METHOD CREATE_JOB : BOOL
VAR_INPUT
	_byMbFunction	:	BYTE;
	_wMbAdress		:	WORD;
	_pData			:	POINTER TO BYTE;
	_wQuantity		:	WORD;		
END_VAR
VAR	
	pFbMbJob		:	POINTER TO FB_MBJOB;
END_VAR
IF _pData <> 0 THEN
	IF NOT CHECK_IF_JOB_EXIST(_byMbFunction,_wMbAdress,_pData,_wQuantity) THEN
		pFbMbJob := __NEW(FB_MBJOB);
		IF pFbMbJob <> 0 THEN
			_udiDynMemTemp 			:= _udiDynMemTemp + SIZEOF(FB_MBJOB);
			udiDynMem				:= MAX(udiDynMem,_udiDynMemTemp);
			pFbMbJob^.byMbFunction 	:= _byMbFunction;
			pFbMbJob^.wMbAdress	 	:= _wMbAdress;
			pFbMbJob^.pByte		 	:= _pData;
			pFbMbJob^.wQuantity 	:= _wQuantity;
			ADD_MODBUS_JOB(pFbMbJob^);
			xNoChangeHappen			:= FALSE;
			xConfirmAllJobsDone		:= FALSE;
		END_IF;
	END_IF;
END_IF;
END_METHOD

METHOD DESTROY_JOB : BOOL
VAR_INPUT
	_byMbFunction	:	BYTE;
	_wMbAdress		:	WORD;
	_pData			:	POINTER TO BYTE;
	_wQuantity		:	WORD;		
END_VAR
VAR	
	udiSafe			:	UDINT;
	_TEMP_DES_JOB	:	ITF_MBJOB;
END_VAR
IF __QUERYINTERFACE(_BASE_MBU_JOB,_TEMP_DES_JOB) THEN
	REPEAT 
		IF _TEMP_DES_JOB.byMbFunction = _byMbFunction AND
			_TEMP_DES_JOB.wMbAdress	= _wMbAdress AND
			_TEMP_DES_JOB.pByte = _pData AND
			_TEMP_DES_JOB.wQuantity = _wQuantity THEN
			IF _TEMP_DES_JOB = _TEMP_REG_JOB THEN
				_TEMP_REG_JOB := _TEMP_DES_JOB.BIG_SYBIL;
			END_IF;
			IF _TEMP_DES_JOB = _BASE_MBU_JOB THEN
				_BASE_MBU_JOB := _TEMP_DES_JOB.LOW_SYBIL;
				IF NOT __QUERYINTERFACE(_BASE_MBU_JOB,_BASE_MBU_JOB) THEN
					_TEMP_REG_JOB := _BASE_MBU_JOB;
				END_IF;
			END_IF;
			_TEMP_DES_JOB.DESTROY();
			_COUNT 			:= _COUNT -1;
			_udiDynMemTemp 	:= _udiDynMemTemp - SIZEOF(FB_MBJOB);
			DESTROY_JOB 	:= TRUE;
		ELSE
			_TEMP_DES_JOB := _TEMP_DES_JOB.LOW_SYBIL;
		END_IF;
		udiSafe	:= udiSafe + 1;
	UNTIL DESTROY_JOB OR _TEMP_DES_JOB = 0 OR udiSafe >= 16#FFFFFFFE
	END_REPEAT
ELSE
	DESTROY_JOB := FALSE;
END_IF
END_METHOD

PROPERTY ERROR : BOOL
GET
ERROR := xErrorHappen;
END_GET
SET
xErrorHappen := ERROR;
END_SET
END_PROPERTY

{attribute 'estimated-stack-usage' := '104'}
PROPERTY BIG_SYBIL : ITF_CLIENT
GET
BIG_SYBIL := _ITF_BIG_SYBIL;
END_GET
SET
_ITF_BIG_SYBIL := BIG_SYBIL;
IF __QUERYINTERFACE(_ITF_BIG_SYBIL,_ITF_BIG_SYBIL) THEN
	IF _ITF_BIG_SYBIL.LOW_SYBIL <> SELF THEN
		_ITF_BIG_SYBIL.LOW_SYBIL := THIS^;
	END_IF;
END_IF;
END_SET
END_PROPERTY

METHOD CALL_AFTER_LAST_JOB_DONE
VAR_INPUT
END_VAR
xConfirmAllJobsDone := xNoChangeHappen;
xGetReadyCalled := FALSE;
IF xDestroyAllJobs THEN
	DESTROY_ALL_JOBS();
	xDestroyAllJobs := FALSE;
END_IF;
END_METHOD

METHOD CHECK_IF_JOB_EXIST : BOOL
VAR_INPUT
	_byMbFunction	:	BYTE;
	_wMbAdress		:	WORD;
	_pByte			:	POINTER TO BYTE;
	_wQuantity		:	WORD;	
END_VAR
VAR
	_TEMP_CHK_JOB	:	ITF_MBJOB;
	udiSafe			:	UDINT;
END_VAR
IF __QUERYINTERFACE(_BASE_MBU_JOB,_TEMP_CHK_JOB) THEN
	REPEAT 
		IF _TEMP_CHK_JOB.byMbFunction = _byMbFunction AND
			_TEMP_CHK_JOB.wMbAdress	= _wMbAdress AND
			_TEMP_CHK_JOB.pByte = _pByte AND
			_TEMP_CHK_JOB.wQuantity = _wQuantity THEN
			CHECK_IF_JOB_EXIST := TRUE;
		END_IF;
		_TEMP_CHK_JOB := _TEMP_CHK_JOB.LOW_SYBIL;
		udiSafe	:= udiSafe + 1;
	UNTIL CHECK_IF_JOB_EXIST OR _TEMP_CHK_JOB = 0 OR udiSafe >= 16#FFFFFFFE
	END_REPEAT
ELSE
	CHECK_IF_JOB_EXIST := FALSE;
END_IF
END_METHOD

PROPERTY CONFIRM_ALL_JOBS_DONE : BOOL
GET
CONFIRM_ALL_JOBS_DONE := xConfirmAllJobsDone;
END_GET
END_PROPERTY

PROPERTY AllJobsDone : BOOL
GET
AllJobsDone := xAllJobsDone;
END_GET
END_PROPERTY

PROPERTY AY_ITF_MBJOB_VIS : ARRAY[0..9] OF ITF_MBJOB
GET
AY_ITF_MBJOB_VIS := _ayITF_MBJOB_VIS;
END_GET
END_PROPERTY

PROPERTY BASE_MBJOB : ITF_MBJOB
GET
BASE_MBJOB := _BASE_MBU_JOB;
END_GET
END_PROPERTY

PROPERTY ERROR_ID : ModbusFB.Error
GET
ERROR_ID := eErrorID;
END_GET
SET
eErrorID := ERROR_ID;
END_SET
END_PROPERTY

PROPERTY ExecuteTime : LTIME
GET
ExecuteTime := ltTime;
END_GET
END_PROPERTY

PROPERTY EXEPTION_CODE : ModbusFB.ExceptionCodes
GET
EXEPTION_CODE := eExeptionCode;
END_GET
SET
eExeptionCode := EXEPTION_CODE;
END_SET
END_PROPERTY

METHOD GET_NEXT_JOB : BOOL
VAR_OUTPUT
	_byMbFunction	:	BYTE;
	_wMbAdress		:	WORD;
	_pByte			:	POINTER TO BYTE;
	_wQuantity		:	WORD;	
END_VAR
IF xGetReadyCalled THEN 
	IF __QUERYINTERFACE(_TEMP_MBU_JOB,_TEMP_MBU_JOB) THEN
		_byMbFunction		:= _TEMP_MBU_JOB.byMbFunction;
		_wMbAdress			:= _TEMP_MBU_JOB.wMbAdress;
		_pByte				:= _TEMP_MBU_JOB.pByte;
		_wQuantity			:= _TEMP_MBU_JOB.wQuantity;	
		_TEMP_MBU_JOB		:= _TEMP_MBU_JOB.LOW_SYBIL;
		GET_NEXT_JOB		:= TRUE;
		IF NOT __QUERYINTERFACE(_TEMP_MBU_JOB,_TEMP_MBU_JOB) THEN
			xAllJobsDone 	:= TRUE;
			ltTime			:= fbTimeStop.Stop();
		END_IF;
	ELSIF  __QUERYINTERFACE(_BASE_MBU_JOB,_TEMP_MBU_JOB) THEN 	
		_byMbFunction		:= _TEMP_MBU_JOB.byMbFunction;
		_wMbAdress			:= _TEMP_MBU_JOB.wMbAdress;
		_pByte				:= _TEMP_MBU_JOB.pByte;
		_wQuantity			:= _TEMP_MBU_JOB.wQuantity;
		_TEMP_MBU_JOB		:= _TEMP_MBU_JOB.LOW_SYBIL;
		GET_NEXT_JOB    	:= TRUE;
		fbTimeStop.Start();
	END_IF;
END_IF;
END_METHOD

METHOD GET_READY : BOOL
VAR_INPUT
END_VAR
xGetReadyCalled := TRUE;
xNoChangeHappen := TRUE;
xAllJobsDone	:= FALSE;
_TEMP_MBU_JOB   := 0;
END_METHOD

PROPERTY IsCurrentCall : BOOL
GET
IsCurrentCall := xGetReadyCalled;
END_GET
END_PROPERTY

{attribute 'estimated-stack-usage' := '104'}
PROPERTY LOW_SYBIL : ITF_CLIENT
GET
LOW_SYBIL := _ITF_LOW_SYBIL;
END_GET
SET
_ITF_LOW_SYBIL := LOW_SYBIL;
IF __QUERYINTERFACE(_ITF_LOW_SYBIL,_ITF_LOW_SYBIL) THEN
	IF _ITF_LOW_SYBIL.BIG_SYBIL <> SELF THEN
		_ITF_LOW_SYBIL.BIG_SYBIL := THIS^;
	END_IF;
END_IF;
END_SET
END_PROPERTY

METHOD RELOAD_ARRAY
VAR_INPUT
	xInit				:	BOOL;
	xLoadNext10			:	BOOL;
	xLoadLast10			:	BOOL;
END_VAR
VAR
	diFor				:	DINT;
	ITF_TEMP_MBJOB_VIS	:	ITF_MBJOB;
	ITF_TEMP_SAFE		:	ITF_MBJOB;
	ITF_TEMP_LAST_VALID	:	ITF_MBJOB;
END_VAR
(* Init Array *)
IF xInit THEN
	_ayITF_MBJOB_VIS[LOWER_BOUND(_ayITF_MBJOB_VIS,1)] := _BASE_MBU_JOB;
	FOR diFor := LOWER_BOUND(_ayITF_MBJOB_VIS,1) TO UPPER_BOUND(_ayITF_MBJOB_VIS,1) -1 DO
		IF __QUERYINTERFACE(_ayITF_MBJOB_VIS[diFor],ITF_TEMP_MBJOB_VIS) THEN
			_ayITF_MBJOB_VIS[diFor + 1]	:= _ayITF_MBJOB_VIS[diFor].LOW_SYBIL;
		ELSE
			_ayITF_MBJOB_VIS[diFor + 1] := 0;
		END_IF;	
	END_FOR;
(* Load Next 10 *)
ELSIF xLoadNext10 THEN
	IF __QUERYINTERFACE(_ayITF_MBJOB_VIS[UPPER_BOUND(_ayITF_MBJOB_VIS,1)],ITF_TEMP_MBJOB_VIS) THEN
		_ayITF_MBJOB_VIS[LOWER_BOUND(_ayITF_MBJOB_VIS,1)] := ITF_TEMP_MBJOB_VIS.LOW_SYBIL;
		FOR diFor := LOWER_BOUND(_ayITF_MBJOB_VIS,1) TO UPPER_BOUND(_ayITF_MBJOB_VIS,1) -1 DO
			IF __QUERYINTERFACE(_ayITF_MBJOB_VIS[diFor],ITF_TEMP_MBJOB_VIS) THEN
				_ayITF_MBJOB_VIS[diFor + 1]	:= _ayITF_MBJOB_VIS[diFor].LOW_SYBIL;
			ELSE
				_ayITF_MBJOB_VIS[diFor + 1] := 0;
			END_IF;	
		END_FOR;
	END_IF;
(* Load Last 10 *)
ELSIF xLoadLast10 THEN
	IF __QUERYINTERFACE(_ayITF_MBJOB_VIS[LOWER_BOUND(_ayITF_MBJOB_VIS,1)],ITF_TEMP_MBJOB_VIS) THEN
		IF __QUERYINTERFACE(_ayITF_MBJOB_VIS[LOWER_BOUND(_ayITF_MBJOB_VIS,1)].BIG_SYBIL,ITF_TEMP_SAFE) THEN
			_ayITF_MBJOB_VIS[UPPER_BOUND(_ayITF_MBJOB_VIS,1)] := ITF_TEMP_MBJOB_VIS.BIG_SYBIL;
			FOR diFor := UPPER_BOUND(_ayITF_MBJOB_VIS,1) TO LOWER_BOUND(_ayITF_MBJOB_VIS,1) + 1 BY -1 DO 
				IF __QUERYINTERFACE(_ayITF_MBJOB_VIS[diFor],ITF_TEMP_MBJOB_VIS) THEN
					ITF_TEMP_LAST_VALID  		:= _ayITF_MBJOB_VIS[diFor];
					_ayITF_MBJOB_VIS[diFor - 1]	:= _ayITF_MBJOB_VIS[diFor].BIG_SYBIL;
				ELSE
					(* Resort if new ones Inside *)
					_ayITF_MBJOB_VIS[LOWER_BOUND(_ayITF_MBJOB_VIS,1)] := ITF_TEMP_LAST_VALID;
					FOR diFor := LOWER_BOUND(_ayITF_MBJOB_VIS,1) TO UPPER_BOUND(_ayITF_MBJOB_VIS,1) -1 DO
						IF __QUERYINTERFACE(_ayITF_MBJOB_VIS[diFor],ITF_TEMP_MBJOB_VIS) THEN
							_ayITF_MBJOB_VIS[diFor + 1]	:= _ayITF_MBJOB_VIS[diFor].LOW_SYBIL;
						ELSE
							_ayITF_MBJOB_VIS[diFor + 1] := 0;
						END_IF;	
					END_FOR;					
				END_IF;	
			END_FOR;
		END_IF;
	END_IF;	
END_IF;
END_METHOD

PROPERTY SELF : ITF_CLIENT
GET
SELF := THIS^;
END_GET
END_PROPERTY

METHOD DESTROY_ALL_JOBS_REQUEST
VAR_INPUT
END_VAR
xDestroyAllJobs := TRUE;
END_METHOD

PROPERTY DESTROY_ALL_JOBS_ACTIVE : BOOL
GET
DESTROY_ALL_JOBS_ACTIVE := xDestroyAllJobs;
END_GET
END_PROPERTY

METHOD INTERNAL DESTROY_ALL_JOBS
VAR_INPUT
END_VAR
VAR
	_TEMP_DES_JOB	:	ITF_MBJOB;
	_NEXT_DES_JOB	:	ITF_MBJOB;
	udiSafe			:	UDINT;
END_VAR
IF __QUERYINTERFACE(_BASE_MBU_JOB,_NEXT_DES_JOB) THEN
	_BASE_MBU_JOB := 0;
	_TEMP_REG_JOB := 0;
	_TEMP_MBU_JOB := 0;
	REPEAT 
		IF __QUERYINTERFACE(_NEXT_DES_JOB, _TEMP_DES_JOB) THEN
			_NEXT_DES_JOB := _TEMP_DES_JOB.LOW_SYBIL;
			_TEMP_DES_JOB.DESTROY();
			_COUNT 			:= _COUNT -1;
			_udiDynMemTemp 	:= _udiDynMemTemp - SIZEOF(FB_MBJOB);
		END_IF;
		udiSafe	:= udiSafe + 1;
	UNTIL _NEXT_DES_JOB = 0 OR udiSafe >= 16#FFFFFFFE
	END_REPEAT
END_IF;
END_METHOD

END_FUNCTION_BLOCK

// 30 Program Organization Units/MBJOB/FB_MBJOB
{attribute 'enable_dynamic_creation'}
FUNCTION_BLOCK FB_MBJOB IMPLEMENTS ITF_MBJOB
VAR_OUTPUT
END_VAR
VAR
	_xConfirmExecute:	BOOL;
	_byMbFunction	:	BYTE;
	_wMbAdress		:	WORD;
	_pByte			:	POINTER TO BYTE;
	_wQuantity		:	WORD;	
	_ITF_BIG_SYBIL	:	ITF_MBJOB;
	_ITF_LOW_SYBIL	:	ITF_MBJOB;
	_ITF_PARENT		:	ITF_CLIENT;
END_VAR

PROPERTY wMbAdress : WORD
GET
wMbAdress := _wMbAdress;
END_GET
SET
_wMbAdress := wMbAdress;
END_SET
END_PROPERTY

{attribute 'estimated-stack-usage' := '104'}
PROPERTY BIG_SYBIL : ITF_MBJOB
GET
BIG_SYBIL := _ITF_BIG_SYBIL;
END_GET
SET
_ITF_BIG_SYBIL := BIG_SYBIL;
IF __QUERYINTERFACE(_ITF_BIG_SYBIL,_ITF_BIG_SYBIL) THEN
	IF _ITF_BIG_SYBIL.LOW_SYBIL <> SELF THEN
		_ITF_BIG_SYBIL.LOW_SYBIL := THIS^;
	END_IF;
END_IF;
END_SET
END_PROPERTY

PROPERTY wQuantity : WORD
GET
wQuantity := _wQuantity;
END_GET
SET
_wQuantity := wQuantity;
END_SET
END_PROPERTY

PROPERTY SELF : ITF_MBJOB
GET
SELF := THIS^;
END_GET
END_PROPERTY

PROPERTY byMbFunction : BYTE
SET
_byMbFunction := byMbFunction;
END_SET
GET
byMbFunction := _byMbFunction;
END_GET
END_PROPERTY

METHOD DESTROY
VAR
	pSelf	:	POINTER TO FB_MBJOB;
END_VAR
IF __QUERYINTERFACE(_ITF_BIG_SYBIL,_ITF_BIG_SYBIL) THEN
	_ITF_BIG_SYBIL.LOW_SYBIL := _ITF_LOW_SYBIL;
END_IF;

IF __QUERYINTERFACE(_ITF_LOW_SYBIL,_ITF_LOW_SYBIL) THEN
	_ITF_LOW_SYBIL.BIG_SYBIL := _ITF_BIG_SYBIL;
END_IF;

IF __QUERYINTERFACE(_ITF_PARENT,_ITF_PARENT) THEN
	_ITF_PARENT.RELOAD_ARRAY(TRUE,FALSE,FALSE);
END_IF;

pSelf := THIS;

__DELETE(pSelf);
END_METHOD

{attribute 'estimated-stack-usage' := '104'}
PROPERTY LOW_SYBIL : ITF_MBJOB
SET
_ITF_LOW_SYBIL := LOW_SYBIL;
IF __QUERYINTERFACE(_ITF_LOW_SYBIL,_ITF_LOW_SYBIL) THEN
	IF _ITF_LOW_SYBIL.BIG_SYBIL <> SELF THEN
		_ITF_LOW_SYBIL.BIG_SYBIL := THIS^;
	END_IF;
END_IF;
END_SET
GET
LOW_SYBIL := _ITF_LOW_SYBIL;
END_GET
END_PROPERTY

PROPERTY PARENT : ITF_CLIENT
SET
_ITF_PARENT := PARENT;
END_SET
END_PROPERTY

PROPERTY pByte : POINTER TO BYTE
SET
_pByte := pByte;
END_SET
GET
pByte := _pByte;
END_GET
END_PROPERTY

END_FUNCTION_BLOCK

// 30 Program Organization Units/CLIENTMANAGER/RTU/FB_MB_CLIENTMANAGER_RTU
{attribute 'no_assign'}
FUNCTION_BLOCK FB_MB_CLIENTMANAGER_RTU EXTENDS FB_MB_CLIENTMANAGER IMPLEMENTS ITF_MB_CLIENTMANAGER_RTU
VAR_OUTPUT
END_VAR
VAR
	Client								:	ModbusFB.ClientSerial;
	
	_TEMP_MBU_CLIENT_RTU				:	ITF_MB_CLIENT_RTU;
	
	fbReadCoilsFc01						:	ModbusFB.ClientRequestReadCoils;
	fbReadDiscreteInputsFc02			:	ModbusFB.ClientRequestReadDiscreteInputs;
	fbReadHoldingRegistersFc03			:	ModbusFB.ClientRequestReadHoldingRegisters;
	fbReadInputRegistersFc04			:	ModbusFB.ClientRequestReadInputRegisters;
	fbWriteSingleCoilFc05				:	ModbusFB.ClientRequestWriteSingleCoil;
	fbWriteSingleRegisterFc06			:	ModbusFB.ClientRequestWriteSingleRegister;
	fbWriteMultipleCoilsFc15			:	ModbusFB.ClientRequestWriteMultipleCoils;
	fbWriteMultipleRegistersFc16		:	ModbusFB.ClientRequestWriteMultipleRegisters;
	
	(*Config File *)
	fbConfigFile						:	CtaSysConfig.fbConfigFile;
	scParameter                	 		: 	scSerialPortParameter;
END_VAR

SUPER^();
(* Config *)
actConfig();
(* Check if one is allready Working *)
IF NOT xIsWorking THEN
	(* Get Client Ready *)
	IF __QUERYINTERFACE(_TEMP_MBU_CLIENT,_TEMP_MBU_CLIENT) THEN
		xIsWorking 		:= TRUE;	
		xErrorHappen	:= FALSE;
		eErrorID		:= ModbusFB.Error.OK;
		eExeptionCode	:= ModbusFB.ExceptionCodes.RESPONSE_SUCCESS;	
	(* Get Base Client Ready *)
	ELSIF __QUERYINTERFACE(_BASE_MBU_CLIENT,_TEMP_MBU_CLIENT) THEN
		xIsWorking 		:= TRUE;
		xErrorHappen	:= FALSE;
		eErrorID		:= ModbusFB.Error.OK;
		eExeptionCode	:= ModbusFB.ExceptionCodes.RESPONSE_SUCCESS;
		ltTime := fbTimeStop.Stop();
		fbTimeStop.Start();
	END_IF;
END_IF;
(* Check if is running *)
IF xIsWorking THEN
	IF __QUERYINTERFACE(_TEMP_MBU_CLIENT,_TEMP_MBU_CLIENT) THEN	
		(* Wait until no Execute *)		
		IF 	NOT	fbReadCoilsFc01.xExecute				AND
			NOT	fbReadDiscreteInputsFc02.xExecute	    AND
			NOT	fbReadHoldingRegistersFc03.xExecute     AND
			NOT	fbReadInputRegistersFc04.xExecute	    AND
			NOT	fbWriteSingleCoilFc05.xExecute		    AND
			NOT	fbWriteSingleRegisterFc06.xExecute	    AND
			NOT	fbWriteMultipleCoilsFc15.xExecute	    AND
			NOT	fbWriteMultipleRegistersFc16.xExecute	THEN
			(* Get Type of Port *) 
			IF __QUERYINTERFACE(_TEMP_MBU_CLIENT,_TEMP_MBU_CLIENT_RTU) THEN
				(* Check if Enabled *)
				IF _TEMP_MBU_CLIENT_RTU.ENABLE AND _TEMP_MBU_CLIENT_RTU.COUNT > 0 THEN
					IF NOT _TEMP_MBU_CLIENT_RTU.IsCurrentCall THEN
						_TEMP_MBU_CLIENT_RTU.GET_READY();
					END_IF;
					(* Connect *)
					IF NOT Client.xConnected THEN
						Client.xConnect		:= TRUE;
						Client.iPort		:= scParameter.fbenPort.proValue;
						Client.dwBaudrate	:= scParameter.fbdwBaudrate.proValue;
						Client.byDataBits	:= scParameter.fbbyDataBits.proValue;
						Client.eParity		:= scParameter.fbenParity.proValue;
						Client.eStopBits	:= scParameter.fbenStopBits.proValue;
						Client.eDTRcontrol	:= scParameter.fbenDTRControl.proValue;
						Client.eRTScontrol	:= scParameter.fbenRTSControl.proValue;
						IF scParameter.fbxRtuAscii.proValue THEN
							Client.eRtuAscii	:= ModbusFB.RtuAscii.ASCII;
						ELSE
							Client.eRtuAscii	:= ModbusFB.RtuAscii.RTU;
						END_IF
					END_IF;
					usiNodeId 			:= _TEMP_MBU_CLIENT_RTU.NODE_ID;
					tTimeOut			:= _TEMP_MBU_CLIENT_RTU.TIMEOUT;
					tReadDelay			:= _TEMP_MBU_CLIENT_RTU.READ_DELAY;
					tWriteDelay	 		:= _TEMP_MBU_CLIENT_RTU.WRITE_DELAY;
				ELSE
					xAbort		:= TRUE;
				END_IF;
			ELSE
				xAbort		:= TRUE;				
			END_IF;
			(* Check if Connected *)
			IF Client.xConnected AND NOT xAbort THEN
				(* Get Job *)
				IF NOT xTrig THEN
					xTrig := _TEMP_MBU_CLIENT.GET_NEXT_JOB(_byMbFunction => _byMbFunction,_wMbAdress => _wMbAdress,_pByte => _pByte,_wQuantity => _wQuantity);
				END_IF;
				
				(* Delay Function *)
				actDelays();
				
				(* Execute Function *)
				actExecuteFunction();
				
				(* Resett Timer *)
				IF tonDelay.Q THEN
					tonDelay(IN := FALSE);
					xTrig := FALSE;
				END_IF;
			END_IF;
		ELSE
			(* Check Busy *)
			actCheckBusy();					
		END_IF;
		(* Get Errors *)
		actGetError();
		(* Check if All Job as Done *)
		IF _TEMP_MBU_CLIENT.AllJobsDone OR xAbort THEN
			(* Wait until no Execute *)		
			IF 	NOT xTrig									AND
				NOT	fbReadCoilsFc01.xExecute				AND
				NOT	fbReadDiscreteInputsFc02.xExecute	    AND
				NOT	fbReadHoldingRegistersFc03.xExecute     AND
				NOT	fbReadInputRegistersFc04.xExecute	    AND
				NOT	fbWriteSingleCoilFc05.xExecute		    AND
				NOT	fbWriteSingleRegisterFc06.xExecute	    AND
				NOT	fbWriteMultipleCoilsFc15.xExecute	    AND
				NOT	fbWriteMultipleRegistersFc16.xExecute	THEN
				_TEMP_MBU_CLIENT.CALL_AFTER_LAST_JOB_DONE();
				(* Set Error if Job > 0 *)
				IF _TEMP_MBU_CLIENT.COUNT > 0 THEN
					_TEMP_MBU_CLIENT.ERROR			:= xErrorHappen;
					_TEMP_MBU_CLIENT.ERROR_ID		:= eErrorID;
					_TEMP_MBU_CLIENT.EXEPTION_CODE	:= eExeptionCode;
				END_IF;
				_TEMP_MBU_CLIENT 				:= _TEMP_MBU_CLIENT.LOW_SYBIL;
				xIsWorking						:= FALSE;
				xAbort							:= FALSE;
				_byMbFunction 					:= 0;
				_wMbAdress	  					:= 0;
				_pByte		  					:= 0;
				_wQuantity						:= 0;
			END_IF;
		END_IF;
	END_IF;
END_IF;

(* Call Functions *)
actCallFunctions();

(* Resett Client on Error *)
IF Client.xError AND Client._xConnect THEN
	Client.xConnect := FALSE;
END_IF
(* Call Client *)
Client(udiLogOptions := ModbusFB.LoggingOptions.ServerExceptionReason);

ACTION actCallFunctions:
(* Call *)
fbReadCoilsFc01(				rClient := client);		
fbReadDiscreteInputsFc02(		rClient := Client);  
fbReadHoldingRegistersFc03(		rClient := Client);
fbReadInputRegistersFc04(		rClient := Client);	  
fbWriteSingleCoilFc05(			rClient := Client);	  
fbWriteSingleRegisterFc06(		rClient := Client);  
fbWriteMultipleCoilsFc15(		rClient := Client);  
fbWriteMultipleRegistersFc16(	rClient := Client);
END_ACTION

ACTION actDelays:
(* Delay Read *)
IF _byMbFunction <= 04 THEN
	tonDelay(IN := xTrig,PT := tReadDelay);
(* Delay Write Single *)
ELSIF _byMbFunction >= 5 AND _byMbFunction <= 6 THEN
	tonDelay(IN := xTrig,PT := tWriteDelay); 
(* Delay Write Multiple *)
ELSIF _byMbFunction >= 15 AND _byMbFunction <= 16 THEN
	tonDelay(IN := xTrig,PT := tWriteDelay); 
ELSE 
	tonDelay(IN := xTrig,PT := T#0MS);
END_IF;
END_ACTION

ACTION actConfig:
fbConfigFile();		
scParameter.fbenPort			(_usiParaNr := 1,itfConfigFb := fbconfigFile , _MinInit :=    0,_MaxInit :=    10);
scParameter.fbdwBaudrate		(_usiParaNr := 2,itfConfigFb := fbconfigFile , _MinInit := 4800,_MaxInit := 115200);
scParameter.fbbyDataBits		(_usiParaNr := 3,itfConfigFb := fbconfigFile , _MinInit :=    0,_MaxInit :=     8);
scParameter.fbenParity			(_usiParaNr := 4,itfConfigFb := fbconfigFile , _MinInit :=    0,_MaxInit :=     2);
scParameter.fbenStopBits		(_usiParaNr := 5,itfConfigFb := fbconfigFile , _MinInit :=    1,_MaxInit :=     3);
scParameter.fbenDTRControl		(_usiParaNr := 6,itfConfigFb := fbconfigFile , _MinInit :=    0,_MaxInit :=     2);
scParameter.fbenRTSControl		(_usiParaNr := 7,itfConfigFb := fbconfigFile , _MinInit :=    0,_MaxInit :=     2);
scParameter.fbxRtuAscii			(_usiParaNr := 8,itfConfigFb := fbconfigFile 								 	);

(* Handle on Change *)
IF scParameter.fbenPort.proStateChanged			OR
   scParameter.fbdwBaudrate.proStateChanged	    OR
   scParameter.fbbyDataBits.proStateChanged	    OR
   scParameter.fbenParity.proStateChanged		OR
   scParameter.fbenStopBits.proStateChanged	    OR
   scParameter.fbenDTRControl.proStateChanged	OR
   scParameter.fbenRTSControl.proStateChanged	OR
   scParameter.fbxRtuAscii.proStateChanged		THEN
   Client.xConnect := FALSE;
END_IF;
END_ACTION

ACTION actExecuteFunction:
(* Read Coils *)
IF _byMbFunction = 01 THEN
	fbReadCoilsFc01.udiReplyTimeout					:= TO_UDINT(tTimeOut) * 1000; 
	fbReadCoilsFc01.udiTimeOut						:= 15000000;
	fbReadCoilsFc01.uiUnitId						:= usiNodeId;
	fbReadCoilsFc01.uiStartItem 					:= TO_UINT(_wMbAdress);
	fbReadCoilsFc01.pData 							:= _pByte;
	fbReadCoilsFc01.uiQuantity						:= TO_UINT(_wQuantity);
	fbReadCoilsFc01.xExecute						:= tonDelay.Q;
(* Read Discret Inputs *)                       	
ELSIF _byMbFunction = 02 THEN                   	
	fbReadDiscreteInputsFc02.udiReplyTimeout		:= TO_UDINT(tTimeOut) * 1000; 
	fbReadDiscreteInputsFc02.udiTimeOut				:= 15000000;
	fbReadDiscreteInputsFc02.uiUnitId				:= usiNodeId;
	fbReadDiscreteInputsFc02.uiStartItem			:= TO_UINT(_wMbAdress);
	fbReadDiscreteInputsFc02.pData 					:= _pByte;
	fbReadDiscreteInputsFc02.uiQuantity				:= TO_UINT(_wQuantity);
	fbReadDiscreteInputsFc02.xExecute				:= tonDelay.Q;
(* Read Holding Registers *)                		
ELSIF _byMbFunction = 03 THEN                   	
	fbReadHoldingRegistersFc03.udiReplyTimeout		:= TO_UDINT(tTimeOut) * 1000; 
	fbReadHoldingRegistersFc03.udiTimeOut			:= 15000000;
	fbReadHoldingRegistersFc03.uiUnitId				:= usiNodeId;          	
	fbReadHoldingRegistersFc03.uiStartItem			:= TO_UINT(_wMbAdress);
	fbReadHoldingRegistersFc03.pData 				:= _pByte;
	fbReadHoldingRegistersFc03.uiQuantity			:= TO_UINT(_wQuantity);
	fbReadHoldingRegistersFc03.xExecute				:= tonDelay.Q;			
(* Read Input Registers *)	                		
ELSIF _byMbFunction = 04 THEN                   	
	fbReadInputRegistersFc04.udiReplyTimeout		:= TO_UDINT(tTimeOut) * 1000; 
	fbReadInputRegistersFc04.udiTimeOut				:= 15000000;
	fbReadInputRegistersFc04.uiUnitId				:= usiNodeId;               	
	fbReadInputRegistersFc04.uiStartItem 			:= TO_UINT(_wMbAdress);
	fbReadInputRegistersFc04.pData 					:= _pByte;
	fbReadInputRegistersFc04.uiQuantity				:= TO_UINT(_wQuantity);
	fbReadInputRegistersFc04.xExecute				:= tonDelay.Q;			
(* Write Single Coil *)	                    		
ELSIF _byMbFunction = 05 THEN                   	
	fbWriteSingleCoilFc05.udiReplyTimeout			:= TO_UDINT(tTimeOut) * 1000; 
	fbWriteSingleCoilFc05.udiTimeOut				:= 15000000;
	fbWriteSingleCoilFc05.uiUnitId					:= usiNodeId;            	
	fbWriteSingleCoilFc05.uiItem 					:= TO_UINT(_wMbAdress);
	fbWriteSingleCoilFc05.xValue 					:= FcBytePointToBoolValue(_pByte);
	fbWriteSingleCoilFc05.xExecute					:= tonDelay.Q;		
(* Write Single Register *)                 		
ELSIF _byMbFunction = 06 THEN                   	
	fbWriteSingleRegisterFc06.udiReplyTimeout		:= TO_UDINT(tTimeOut) * 1000;    
	fbWriteSingleRegisterFc06.udiTimeOut			:= 15000000; 
	fbWriteSingleRegisterFc06.uiUnitId				:= usiNodeId;           	
	fbWriteSingleRegisterFc06.uiItem	  			:= TO_UINT(_wMbAdress);
	fbWriteSingleRegisterFc06.uiValue 				:= FcBytePointToWordValue(_pByte);
	fbWriteSingleRegisterFc06.xExecute				:= tonDelay.Q;		
(* Write Multiple Coils *)		            		
ELSIF _byMbFunction = 15 THEN                   	
	fbWriteMultipleCoilsFc15.udiReplyTimeout		:= TO_UDINT(tTimeOut) * 1000;
	fbWriteMultipleCoilsFc15.udiTimeOut				:= 15000000;
	fbWriteMultipleCoilsFc15.uiUnitId				:= usiNodeId;              	
	fbWriteMultipleCoilsFc15.uiStartItem 			:= TO_UINT(_wMbAdress);
	fbWriteMultipleCoilsFc15.pData 					:= _pByte;
	fbWriteMultipleCoilsFc15.uiQuantity				:= TO_UINT(_wQuantity);
	fbWriteMultipleCoilsFc15.xExecute				:= tonDelay.Q;
(* Write Multiple Registers *)                  	
ELSIF _byMbFunction = 16 THEN                   	
	fbWriteMultipleRegistersFc16.udiReplyTimeout	:= TO_UDINT(tTimeOut) * 1000; 
	fbWriteMultipleRegistersFc16.udiTimeOut			:= 15000000;
	fbWriteMultipleRegistersFc16.uiUnitId			:= usiNodeId;    
	fbWriteMultipleRegistersFc16.uiStartItem 		:= TO_UINT(_wMbAdress);
	fbWriteMultipleRegistersFc16.pData 				:= _pByte;
	fbWriteMultipleRegistersFc16.uiQuantity			:= TO_UINT(_wQuantity);
	fbWriteMultipleRegistersFc16.xExecute			:= tonDelay.Q;	
END_IF;
END_ACTION

ACTION actGetError:
(* Client Error *)
IF Client.xError THEN
	xErrorHappen 	:= Client.xError;
	eErrorID		:= Client.eErrorID;
	eExeptionCode	:= ModbusFB.ExceptionCodes.ACKNOWLEDGE;
	xAbort			:= TRUE;
END_IF;
(* Read Coils Fc01 Error *)
IF fbReadCoilsFc01.xError AND NOT xErrorHappen THEN
	xErrorHappen 	:= fbReadCoilsFc01.xError;
	eErrorID		:= fbReadCoilsFc01.eErrorID;
	eExeptionCode	:= fbReadCoilsFc01.eException;
END_IF;
(* Read Discrete Inputs Fc02 Error *)
IF fbReadDiscreteInputsFc02.xError AND NOT xErrorHappen THEN
	xErrorHappen 	:= fbReadDiscreteInputsFc02.xError;
	eErrorID		:= fbReadDiscreteInputsFc02.eErrorID;
	eExeptionCode	:= fbReadDiscreteInputsFc02.eException;
END_IF;
(* Read Holding Registers Fc03 Error *)
IF fbReadHoldingRegistersFc03.xError AND NOT xErrorHappen THEN
	xErrorHappen 	:= fbReadHoldingRegistersFc03.xError;
	eErrorID		:= fbReadHoldingRegistersFc03.eErrorID;
	eExeptionCode	:= fbReadHoldingRegistersFc03.eException;
END_IF;
(* Read Input Registers Fc04 Error *)
IF fbReadInputRegistersFc04.xError AND NOT xErrorHappen THEN
	xErrorHappen 	:= fbReadInputRegistersFc04.xError;
	eErrorID		:= fbReadInputRegistersFc04.eErrorID;
	eExeptionCode	:= fbReadInputRegistersFc04.eException;
END_IF;
(* Write Single Coil Fc05 Error *)
IF fbWriteSingleCoilFc05.xError AND NOT xErrorHappen THEN
	xErrorHappen 	:= fbWriteSingleCoilFc05.xError;
	eErrorID		:= fbWriteSingleCoilFc05.eErrorID;
	eExeptionCode	:= fbWriteSingleCoilFc05.eException;
END_IF;
(* Write Single Register Fc06 Error *)
IF fbWriteSingleRegisterFc06.xError AND NOT xErrorHappen THEN
	xErrorHappen 	:= fbWriteSingleRegisterFc06.xError;
	eErrorID		:= fbWriteSingleRegisterFc06.eErrorID;
	eExeptionCode	:= fbWriteSingleRegisterFc06.eException;
END_IF;		
(* Write Multiple Coils Fc15 Error *)
IF fbWriteMultipleCoilsFc15.xError AND NOT xErrorHappen THEN
	xErrorHappen 	:= fbWriteMultipleCoilsFc15.xError;
	eErrorID		:= fbWriteMultipleCoilsFc15.eErrorID;
	eExeptionCode	:= fbWriteMultipleCoilsFc15.eException;
END_IF;
(* Write Multiple Registers Fc16 Error *)
IF fbWriteMultipleRegistersFc16.xError AND NOT xErrorHappen THEN
	xErrorHappen 	:= fbWriteMultipleRegistersFc16.xError;
	eErrorID		:= fbWriteMultipleRegistersFc16.eErrorID;
	eExeptionCode	:= fbWriteMultipleRegistersFc16.eException;
END_IF;
END_ACTION

PROPERTY P_fbbyDataBits : CtaSysConfig.ITF_DATATYPE
GET
P_fbbyDataBits := scParameter.fbbyDataBits;
END_GET
END_PROPERTY

PROPERTY P_fbdwBaudrate : CtaSysConfig.ITF_DATATYPE
GET
P_fbdwBaudrate := scParameter.fbdwBaudrate;
END_GET
END_PROPERTY

PROPERTY P_fbenDTRControl : CtaSysConfig.ITF_BYTE
GET
P_fbenDTRControl := scParameter.fbenDTRControl;
END_GET
END_PROPERTY

PROPERTY P_fbenParity : CtaSysConfig.ITF_BYTE
GET
P_fbenParity := scParameter.fbenParity;
END_GET
END_PROPERTY

PROPERTY P_fbenRTSControl : CtaSysConfig.ITF_BYTE
GET
P_fbenRTSControl := scParameter.fbenRTSControl;
END_GET
END_PROPERTY

PROPERTY P_fbenStopBits : CtaSysConfig.ITF_BYTE
GET
P_fbenStopBits := scParameter.fbenStopBits;
END_GET
END_PROPERTY

PROPERTY P_fbxRtuAscii : CtaSysConfig.ITF_DATATYPE
GET
P_fbxRtuAscii := scParameter.fbxRtuAscii;
END_GET
END_PROPERTY

PROPERTY P_fbenPort : CtaSysConfig.ITF_INT
GET
P_fbenPort := scParameter.fbenPort;
END_GET
END_PROPERTY

ACTION actCheckBusy:
(* Reset after Busy *)
fbReadCoilsFc01.xExecute				:= fbReadCoilsFc01.xBusy				;
fbReadDiscreteInputsFc02.xExecute	    := fbReadDiscreteInputsFc02.xBusy		;
fbReadHoldingRegistersFc03.xExecute     := fbReadHoldingRegistersFc03.xBusy		;
fbReadInputRegistersFc04.xExecute	    := fbReadInputRegistersFc04.xBusy		;
fbWriteSingleCoilFc05.xExecute		    := fbWriteSingleCoilFc05.xBusy			;
fbWriteSingleRegisterFc06.xExecute	    := fbWriteSingleRegisterFc06.xBusy		;
fbWriteMultipleCoilsFc15.xExecute	    := fbWriteMultipleCoilsFc15.xBusy		;
fbWriteMultipleRegistersFc16.xExecute   := fbWriteMultipleRegistersFc16.xBusy	;
END_ACTION

END_FUNCTION_BLOCK

// 30 Program Organization Units/CLIENT/RTU/FB_MB_CLIENT_RTU
FUNCTION_BLOCK FB_MB_CLIENT_RTU EXTENDS FB_MB_CLIENT IMPLEMENTS ITF_MB_CLIENT_RTU
VAR_OUTPUT
END_VAR
VAR
	(* Config *)
	fbConfigFile				:	CtaSysConfig.fbConfigFile;
	scParameter					:	scSerialClientParameter;
END_VAR

(* Config File *)
actConfig();

ACTION actConfig:
(* Config File *)
fbConfigFile();

scParameter.fbxEnable		(_usiParaNr := 1,itfConfigFb := fbConfigFile										);		
scParameter.fbusiNodeId		(_usiParaNr := 2,itfConfigFb := fbConfigFile,_MinInit := 0	 , _MaxInit := 247		);		
scParameter.fbtTimeOut		(_usiParaNr := 3,itfConfigFb := fbConfigFile,_MinInit := T#0MS, _MaxInit := T#5M 	);		
scParameter.fbtReadDelay	(_usiParaNr := 4,itfConfigFb := fbConfigFile,_MinInit := T#0MS, _MaxInit := T#5M 	);		
scParameter.fbtWriteDelay	(_usiParaNr := 5,itfConfigFb := fbConfigFile,_MinInit := T#0MS, _MaxInit := T#5M 	);
END_ACTION

PROPERTY ENABLE : BOOL
GET
ENABLE := scParameter.fbxEnable.proValue;
END_GET
END_PROPERTY

PROPERTY NODE_ID : USINT
GET
NODE_ID := scParameter.fbusiNodeId.proValue;
END_GET
END_PROPERTY

PROPERTY P_fbtReadDelay : CtaSysConfig.ITF_DATATYPE
GET
P_fbtReadDelay := scParameter.fbtReadDelay;
END_GET
END_PROPERTY

PROPERTY P_fbtTimeOut : CtaSysConfig.ITF_DATATYPE
GET
P_fbtTimeOut := scParameter.fbtTimeOut;
END_GET
END_PROPERTY

PROPERTY P_fbtWriteDelay : CtaSysConfig.ITF_DATATYPE
GET
P_fbtWriteDelay := scParameter.fbtWriteDelay;
END_GET
END_PROPERTY

PROPERTY P_fbusiNodeId : CtaSysConfig.ITF_DATATYPE
GET
P_fbusiNodeId := scParameter.fbusiNodeId;
END_GET
END_PROPERTY

PROPERTY P_fbxEnable : CtaSysConfig.ITF_DATATYPE
GET
P_fbxEnable := scParameter.fbxEnable;
END_GET
END_PROPERTY

PROPERTY READ_DELAY : TIME
GET
READ_DELAY := scParameter.fbtReadDelay.proValue;
END_GET
END_PROPERTY

PROPERTY TIMEOUT : TIME
GET
TIMEOUT := scParameter.fbtTimeOut.proValue;
END_GET
END_PROPERTY

PROPERTY WRITE_DELAY : TIME
GET
WRITE_DELAY := scParameter.fbtWriteDelay.proValue;
END_GET
END_PROPERTY

END_FUNCTION_BLOCK

// 30 Program Organization Units/CLIENT/TCP/FB_MB_CLIENT_TCP
{attribute 'no_assign'}
FUNCTION_BLOCK FB_MB_CLIENT_TCP EXTENDS FB_MB_CLIENT IMPLEMENTS ITF_MB_CLIENT_TCP
VAR_OUTPUT
END_VAR
VAR
	Client						:	ModbusFB.ClientTCP;
	(* Config *)
	fbConfigFile				:	CtaSysConfig.fbConfigFile;
	scParameter                	: 	scTcpClientParameter;
END_VAR

(* Config File *)
actConfig();

(* Resett Client on Error *)
IF (Client.xError AND Client._xConnect) 
	OR NOT ENABLE
	OR scParameter.fbxEnable.proStateChanged		
	OR scParameter.fbuiPort.proStateChanged		
	OR scParameter.fbstIpAdress.proStateChanged	THEN
	Client.xConnect := FALSE;
END_IF

(* Call Client *)
Client(tConnnectTimeOut := T#5S,udiLogOptions := ModbusFB.LoggingOptions.ServerExceptionReason);

ACTION actConfig:
(* Config File *)
fbConfigFile();

scParameter.fbxEnable		(_usiParaNr := 1,itfConfigFb := fbConfigFile										);		
scParameter.fbusiNodeId		(_usiParaNr := 2,itfConfigFb := fbConfigFile,_MinInit := 0	  , _MaxInit := 255		);		
scParameter.fbtTimeOut		(_usiParaNr := 3,itfConfigFb := fbConfigFile,_MinInit := T#0MS, _MaxInit := T#5M 	);		
scParameter.fbtReadDelay	(_usiParaNr := 4,itfConfigFb := fbConfigFile,_MinInit := T#0MS, _MaxInit := T#5M 	);		
scParameter.fbtWriteDelay	(_usiParaNr := 5,itfConfigFb := fbConfigFile,_MinInit := T#0MS, _MaxInit := T#5M 	);	
scParameter.fbuiPort		(_usiParaNr := 6,itfConfigFb := fbConfigFile										);
scParameter.fbstIpAdress	(_usiParaNr := 7,itfConfigFb := fbConfigFile										);

(* Check Ip *)
IF scParameter.fbstIpAdress.proStateChanged THEN
	IF NOT fcCheckIp(scParameter.fbstIPAdress.proValue) THEN
		fcSetInitialIPString(scParameter.fbstIpAdress);
	END_IF;
END_IF;
END_ACTION

PROPERTY ENABLE : BOOL
GET
ENABLE := scParameter.fbxEnable.proValue;
END_GET
END_PROPERTY

PROPERTY IP_ADRESS : STRING(15)
GET
IP_ADRESS := scParameter.fbstIpAdress.proValue;
END_GET
END_PROPERTY

PROPERTY P_fbtTimeOut : CtaSysConfig.ITF_DATATYPE
GET
P_fbtTimeOut := scParameter.fbtTimeOut;
END_GET
END_PROPERTY

PROPERTY P_fbtWriteDelay : CtaSysConfig.ITF_DATATYPE
GET
P_fbtWriteDelay := scParameter.fbtWriteDelay;
END_GET
END_PROPERTY

PROPERTY P_fbuiPort : CtaSysConfig.ITF_DATATYPE
GET
P_fbuiPort := scParameter.fbuiPort;
END_GET
END_PROPERTY

PROPERTY P_fbusiNodeId : CtaSysConfig.ITF_DATATYPE
GET
P_fbusiNodeId := scParameter.fbusiNodeId;
END_GET
END_PROPERTY

PROPERTY P_fbxEnable : CtaSysConfig.ITF_DATATYPE
GET
P_fbxEnable := scParameter.fbxEnable;
END_GET
END_PROPERTY

PROPERTY WRITE_DELAY : TIME
GET
WRITE_DELAY := scParameter.fbtWriteDelay.proValue;
END_GET
END_PROPERTY

PROPERTY PORT : UINT
GET
PORT := scParameter.fbuiPort.proValue;
END_GET
END_PROPERTY

PROPERTY NODE_ID : USINT
GET
NODE_ID := scParameter.fbusiNodeId.proValue;
END_GET
END_PROPERTY

PROPERTY P_fbstIpAdress : CtaSysConfig.ITF_DATATYPE
GET
P_fbstIpAdress := scParameter.fbstIpAdress;
END_GET
END_PROPERTY

PROPERTY READ_DELAY : TIME
GET
READ_DELAY := scParameter.fbtReadDelay.proValue;
END_GET
END_PROPERTY

PROPERTY P_fbtReadDelay : CtaSysConfig.ITF_DATATYPE
GET
P_fbtReadDelay := scParameter.fbtReadDelay;
END_GET
END_PROPERTY

PROPERTY TIMEOUT : TIME
GET
TIMEOUT := scParameter.fbtTimeOut.proValue;
END_GET
END_PROPERTY

METHOD ConnectTcp : BOOL
VAR_INPUT
END_VAR
IF fcCheckIp(IP_ADRESS) THEN
	Client.uiPort 	:= PORT;
	Client.aIPaddr 	:= fcStringIPtoByteArray(IP_ADRESS);
	Client.xConnect	:= TRUE;
	ConnectTcp 		:= TRUE;
ELSE
	ConnectTcp			:= FALSE;
END_IF;
END_METHOD

PROPERTY Connected : BOOL
GET
Connected := Client.xConnected;
END_GET
END_PROPERTY

PROPERTY ClientTcp : REFERENCE TO ModbusFB.Client
GET
ClientTcp REF= Client;
END_GET
END_PROPERTY

END_FUNCTION_BLOCK

// 30 Program Organization Units/CLIENTMANAGER/TCP/FB_MB_CLIENTMANAGER_TCP_1
{attribute 'no_assign'}
FUNCTION_BLOCK FB_MB_CLIENTMANAGER_TCP_1 EXTENDS FB_MB_CLIENTMANAGER IMPLEMENTS ITF_MB_CLIENTMANAGER_TCP
VAR_OUTPUT
END_VAR
VAR
	Client								:	ModbusFB.ClientTCP;

	_TEMP_MBU_CLIENT_TCP				:	ITF_MB_CLIENT_TCP;
	
	fbReadCoilsFc01						:	ModbusFB.ClientRequestReadCoils;
	fbReadDiscreteInputsFc02			:	ModbusFB.ClientRequestReadDiscreteInputs;
	fbReadHoldingRegistersFc03			:	ModbusFB.ClientRequestReadHoldingRegisters;
	fbReadInputRegistersFc04			:	ModbusFB.ClientRequestReadInputRegisters;
	fbWriteSingleCoilFc05				:	ModbusFB.ClientRequestWriteSingleCoil;
	fbWriteSingleRegisterFc06			:	ModbusFB.ClientRequestWriteSingleRegister;
	fbWriteMultipleCoilsFc15			:	ModbusFB.ClientRequestWriteMultipleCoils;
	fbWriteMultipleRegistersFc16		:	ModbusFB.ClientRequestWriteMultipleRegisters;
	
END_VAR

SUPER^();
(* Check if one is allready Working *)
IF NOT xIsWorking THEN
	(* Get Client Ready *)
	IF __QUERYINTERFACE(_TEMP_MBU_CLIENT,_TEMP_MBU_CLIENT) THEN
		xIsWorking 		:= TRUE;	
		xErrorHappen	:= FALSE;
		eErrorID		:= ModbusFB.Error.OK;
		eExeptionCode	:= ModbusFB.ExceptionCodes.RESPONSE_SUCCESS;		
	(* Get Base Client Ready *)
	ELSIF __QUERYINTERFACE(_BASE_MBU_CLIENT,_TEMP_MBU_CLIENT) THEN
		xIsWorking 		:= TRUE;
		xErrorHappen	:= FALSE;
		eErrorID		:= ModbusFB.Error.OK;
		eExeptionCode	:= ModbusFB.ExceptionCodes.RESPONSE_SUCCESS;
		ltTime 			:= fbTimeStop.Stop();
		fbTimeStop.Start();
	END_IF;
END_IF;
(* Check if is running *)
IF xIsWorking THEN
	IF __QUERYINTERFACE(_TEMP_MBU_CLIENT,_TEMP_MBU_CLIENT) THEN	
		(* Wait until no Execute *)		
		IF 	NOT	fbReadCoilsFc01.xExecute				AND
			NOT	fbReadDiscreteInputsFc02.xExecute	    AND
			NOT	fbReadHoldingRegistersFc03.xExecute     AND
			NOT	fbReadInputRegistersFc04.xExecute	    AND
			NOT	fbWriteSingleCoilFc05.xExecute		    AND
			NOT	fbWriteSingleRegisterFc06.xExecute	    AND
			NOT	fbWriteMultipleCoilsFc15.xExecute	    AND
			NOT	fbWriteMultipleRegistersFc16.xExecute	THEN
			(* Get Type of Port *) 
			IF __QUERYINTERFACE(_TEMP_MBU_CLIENT,_TEMP_MBU_CLIENT_TCP) THEN
				(* Check if Enabled *)
				IF _TEMP_MBU_CLIENT_TCP.ENABLE AND _TEMP_MBU_CLIENT_TCP.COUNT > 0 THEN
					IF NOT _TEMP_MBU_CLIENT_TCP.IsCurrentCall THEN
						_TEMP_MBU_CLIENT_TCP.GET_READY();
						tTimeOut		:= _TEMP_MBU_CLIENT_TCP.TIMEOUT;
						tReadDelay		:= _TEMP_MBU_CLIENT_TCP.READ_DELAY;
						tWriteDelay	 	:= _TEMP_MBU_CLIENT_TCP.WRITE_DELAY;
					END_IF;
					(* Connect *)
					IF NOT Client.xConnected THEN
						IF fcCheckIp(_TEMP_MBU_CLIENT_TCP.IP_ADRESS) THEN
							Client.uiPort 	:= _TEMP_MBU_CLIENT_TCP.PORT;
							Client.aIPaddr 	:= fcStringIPtoByteArray(_TEMP_MBU_CLIENT_TCP.IP_ADRESS);
							Client.xConnect	:= TRUE;
							usiNodeId 		:= _TEMP_MBU_CLIENT_TCP.NODE_ID;
						ELSE
							xAbort := TRUE;
						END_IF;
					END_IF;
				ELSE
					xAbort		:= TRUE;
				END_IF;
			ELSE
				xAbort := TRUE;
			END_IF;
			(* Check if Connected *)
			IF Client.xConnected AND NOT xAbort THEN
				(* Get Job *)
				IF NOT xTrig THEN
					xTrig := _TEMP_MBU_CLIENT.GET_NEXT_JOB(_byMbFunction => _byMbFunction,_wMbAdress => _wMbAdress,_pByte => _pByte,_wQuantity => _wQuantity);
				END_IF;
				
				(* Delay Function *)
				actDelays();
				
				(* Execute Function *)
				actExecuteFunction();
				
				(* Resett Timer *)
				IF tonDelay.Q THEN
					tonDelay(IN := FALSE);
					xTrig := FALSE;
				END_IF;
			END_IF;
		ELSE
			(* Check Busy *)
			actCheckBusy();					
		END_IF;
		(* Get Errors *)
		actGetError();
		(* Check if All Job as Done *)
		IF _TEMP_MBU_CLIENT.AllJobsDone OR xAbort THEN
			(* Wait until no Execute *)		
			IF 	NOT	fbReadCoilsFc01.xExecute				AND
				NOT	fbReadDiscreteInputsFc02.xExecute	    AND
				NOT	fbReadHoldingRegistersFc03.xExecute     AND
				NOT	fbReadInputRegistersFc04.xExecute	    AND
				NOT	fbWriteSingleCoilFc05.xExecute		    AND
				NOT	fbWriteSingleRegisterFc06.xExecute	    AND
				NOT	fbWriteMultipleCoilsFc15.xExecute	    AND
				NOT	fbWriteMultipleRegistersFc16.xExecute	THEN
				_TEMP_MBU_CLIENT.CALL_AFTER_LAST_JOB_DONE();
				(* Set Error if Job > 0 *)
				IF _TEMP_MBU_CLIENT.COUNT > 0 THEN
					_TEMP_MBU_CLIENT.ERROR			:= xErrorHappen;
					_TEMP_MBU_CLIENT.ERROR_ID		:= eErrorID;
					_TEMP_MBU_CLIENT.EXEPTION_CODE	:= eExeptionCode;
				END_IF;
				_TEMP_MBU_CLIENT 					:= _TEMP_MBU_CLIENT.LOW_SYBIL;
				
				IF SUPER^.COUNT_ENABLED() = 1 AND NOT xAbort THEN	
					Client.xConnect := Client.xConnect;
				ELSE
					Client.xConnect				:= FALSE;
				END_IF;
				_byMbFunction 					:= 0;
				_wMbAdress	  					:= 0;
				_pByte		  					:= 0;
				_wQuantity						:= 0;
				xIsWorking						:= FALSE;
				xAbort							:= FALSE;
			END_IF;
		END_IF;
	END_IF;
END_IF;

(* Call Functions *)
actCallFunctions();

(* Resett Client on Error *)
IF Client.xError AND Client._xConnect THEN
	Client.xConnect := FALSE;
END_IF
(* Call Client *)
Client(tConnnectTimeOut := T#5S,udiLogOptions := ModbusFB.LoggingOptions.ServerExceptionReason);

ACTION actCallFunctions:
(* Call *)
fbReadCoilsFc01(				rClient := client);		
fbReadDiscreteInputsFc02(		rClient := Client);  
fbReadHoldingRegistersFc03(		rClient := Client);
fbReadInputRegistersFc04(		rClient := Client);	  
fbWriteSingleCoilFc05(			rClient := Client);	  
fbWriteSingleRegisterFc06(		rClient := Client);  
fbWriteMultipleCoilsFc15(		rClient := Client);  
fbWriteMultipleRegistersFc16(	rClient := Client);
END_ACTION

ACTION actCheckBusy:
(* Reset after Busy *)
fbReadCoilsFc01.xExecute				:= fbReadCoilsFc01.xBusy				;
fbReadDiscreteInputsFc02.xExecute	    := fbReadDiscreteInputsFc02.xBusy		;
fbReadHoldingRegistersFc03.xExecute     := fbReadHoldingRegistersFc03.xBusy		;
fbReadInputRegistersFc04.xExecute	    := fbReadInputRegistersFc04.xBusy		;
fbWriteSingleCoilFc05.xExecute		    := fbWriteSingleCoilFc05.xBusy			;
fbWriteSingleRegisterFc06.xExecute	    := fbWriteSingleRegisterFc06.xBusy		;
fbWriteMultipleCoilsFc15.xExecute	    := fbWriteMultipleCoilsFc15.xBusy		;
fbWriteMultipleRegistersFc16.xExecute   := fbWriteMultipleRegistersFc16.xBusy	;
END_ACTION

ACTION actDelays:
(* Delay Read *)
IF _byMbFunction <= 04 THEN
	tonDelay(IN := xTrig,PT := tReadDelay);
(* Delay Write Single *)
ELSIF _byMbFunction >= 5 AND _byMbFunction <= 6 THEN
	tonDelay(IN := xTrig,PT := tWriteDelay); 
(* Delay Write Multiple *)
ELSIF _byMbFunction >= 15 AND _byMbFunction <= 16 THEN
	tonDelay(IN := xTrig,PT := tWriteDelay); 
ELSE 
	tonDelay(IN := xTrig,PT := T#0MS);
END_IF;
END_ACTION

ACTION actExecuteFunction:
(* Read Coils *)
IF _byMbFunction = 01 THEN
	fbReadCoilsFc01.udiReplyTimeout					:= TO_UDINT(tTimeOut) * 1000; 
	fbReadCoilsFc01.udiTimeOut						:= TO_UDINT(tTimeOut) * 1000 * 2;
	fbReadCoilsFc01.uiUnitId						:= usiNodeId;
	fbReadCoilsFc01.uiStartItem 					:= TO_UINT(_wMbAdress);
	fbReadCoilsFc01.pData 							:= _pByte;
	fbReadCoilsFc01.uiQuantity						:= TO_UINT(_wQuantity);
	fbReadCoilsFc01.xExecute						:= tonDelay.Q;
(* Read Discret Inputs *)                       	
ELSIF _byMbFunction = 02 THEN                   	
	fbReadDiscreteInputsFc02.udiReplyTimeout		:= TO_UDINT(tTimeOut) * 1000; 
	fbReadDiscreteInputsFc02.udiTimeOut				:= TO_UDINT(tTimeOut) * 1000 * 2;
	fbReadDiscreteInputsFc02.uiUnitId				:= usiNodeId;
	fbReadDiscreteInputsFc02.uiStartItem			:= TO_UINT(_wMbAdress);
	fbReadDiscreteInputsFc02.pData 					:= _pByte;
	fbReadDiscreteInputsFc02.uiQuantity				:= TO_UINT(_wQuantity);
	fbReadDiscreteInputsFc02.xExecute				:= tonDelay.Q;
(* Read Holding Registers *)                		
ELSIF _byMbFunction = 03 THEN                   	
	fbReadHoldingRegistersFc03.udiReplyTimeout		:= TO_UDINT(tTimeOut) * 1000; 
	fbReadHoldingRegistersFc03.udiTimeOut			:= TO_UDINT(tTimeOut) * 1000 * 2;
	fbReadHoldingRegistersFc03.uiUnitId				:= usiNodeId;          	
	fbReadHoldingRegistersFc03.uiStartItem			:= TO_UINT(_wMbAdress);
	fbReadHoldingRegistersFc03.pData 				:= _pByte;
	fbReadHoldingRegistersFc03.uiQuantity			:= TO_UINT(_wQuantity);
	fbReadHoldingRegistersFc03.xExecute				:= tonDelay.Q;			
(* Read Input Registers *)	                		
ELSIF _byMbFunction = 04 THEN                   	
	fbReadInputRegistersFc04.udiReplyTimeout		:= TO_UDINT(tTimeOut) * 1000; 
	fbReadInputRegistersFc04.udiTimeOut				:= TO_UDINT(tTimeOut) * 1000 * 2;
	fbReadInputRegistersFc04.uiUnitId				:= usiNodeId;               	
	fbReadInputRegistersFc04.uiStartItem 			:= TO_UINT(_wMbAdress);
	fbReadInputRegistersFc04.pData 					:= _pByte;
	fbReadInputRegistersFc04.uiQuantity				:= TO_UINT(_wQuantity);
	fbReadInputRegistersFc04.xExecute				:= tonDelay.Q;			
(* Write Single Coil *)	                    		
ELSIF _byMbFunction = 05 THEN                   	
	fbWriteSingleCoilFc05.udiReplyTimeout			:= TO_UDINT(tTimeOut) * 1000; 
	fbWriteSingleCoilFc05.udiTimeOut				:= TO_UDINT(tTimeOut) * 1000 * 2;
	fbWriteSingleCoilFc05.uiUnitId					:= usiNodeId;            	
	fbWriteSingleCoilFc05.uiItem 					:= TO_UINT(_wMbAdress);
	fbWriteSingleCoilFc05.xValue 					:= FcBytePointToBoolValue(_pByte);
	fbWriteSingleCoilFc05.xExecute					:= tonDelay.Q;		
(* Write Single Register *)                 		
ELSIF _byMbFunction = 06 THEN                   	
	fbWriteSingleRegisterFc06.udiReplyTimeout		:= TO_UDINT(tTimeOut) * 1000;    
	fbWriteSingleRegisterFc06.udiTimeOut			:= TO_UDINT(tTimeOut) * 1000 * 2; 
	fbWriteSingleRegisterFc06.uiUnitId				:= usiNodeId;           	
	fbWriteSingleRegisterFc06.uiItem	  			:= TO_UINT(_wMbAdress);
	fbWriteSingleRegisterFc06.uiValue 				:= FcBytePointToWordValue(_pByte);
	fbWriteSingleRegisterFc06.xExecute				:= tonDelay.Q;		
(* Write Multiple Coils *)		            		
ELSIF _byMbFunction = 15 THEN                   	
	fbWriteMultipleCoilsFc15.udiReplyTimeout		:= TO_UDINT(tTimeOut) * 1000;
	fbWriteMultipleCoilsFc15.udiTimeOut				:= TO_UDINT(tTimeOut) * 1000 * 2;
	fbWriteMultipleCoilsFc15.uiUnitId				:= usiNodeId;              	
	fbWriteMultipleCoilsFc15.uiStartItem 			:= TO_UINT(_wMbAdress);
	fbWriteMultipleCoilsFc15.pData 					:= _pByte;
	fbWriteMultipleCoilsFc15.uiQuantity				:= TO_UINT(_wQuantity);
	fbWriteMultipleCoilsFc15.xExecute				:= tonDelay.Q;
(* Write Multiple Registers *)                  	
ELSIF _byMbFunction = 16 THEN                   	
	fbWriteMultipleRegistersFc16.udiReplyTimeout	:= TO_UDINT(tTimeOut) * 1000; 
	fbWriteMultipleRegistersFc16.udiTimeOut			:= TO_UDINT(tTimeOut) * 1000 * 2;
	fbWriteMultipleRegistersFc16.uiUnitId			:= usiNodeId;    
	fbWriteMultipleRegistersFc16.uiStartItem 		:= TO_UINT(_wMbAdress);
	fbWriteMultipleRegistersFc16.pData 				:= _pByte;
	fbWriteMultipleRegistersFc16.uiQuantity			:= TO_UINT(_wQuantity);
	fbWriteMultipleRegistersFc16.xExecute			:= tonDelay.Q;	
END_IF;
END_ACTION

ACTION actGetError:
(* Client Error *)
IF Client.xError THEN
	xErrorHappen 	:= Client.xError;
	eErrorID		:= Client.eErrorID;
	eExeptionCode	:= ModbusFB.ExceptionCodes.ACKNOWLEDGE;
	xAbort			:= TRUE;
END_IF;
(* Read Coils Fc01 Error *)
IF fbReadCoilsFc01.xError AND NOT xErrorHappen THEN
	xErrorHappen 	:= fbReadCoilsFc01.xError;
	eErrorID		:= fbReadCoilsFc01.eErrorID;
	eExeptionCode	:= fbReadCoilsFc01.eException;
END_IF;
(* Read Discrete Inputs Fc02 Error *)
IF fbReadDiscreteInputsFc02.xError AND NOT xErrorHappen THEN
	xErrorHappen 	:= fbReadDiscreteInputsFc02.xError;
	eErrorID		:= fbReadDiscreteInputsFc02.eErrorID;
	eExeptionCode	:= fbReadDiscreteInputsFc02.eException;
END_IF;
(* Read Holding Registers Fc03 Error *)
IF fbReadHoldingRegistersFc03.xError AND NOT xErrorHappen THEN
	xErrorHappen 	:= fbReadHoldingRegistersFc03.xError;
	eErrorID		:= fbReadHoldingRegistersFc03.eErrorID;
	eExeptionCode	:= fbReadHoldingRegistersFc03.eException;
END_IF;
(* Read Input Registers Fc04 Error *)
IF fbReadInputRegistersFc04.xError AND NOT xErrorHappen THEN
	xErrorHappen 	:= fbReadInputRegistersFc04.xError;
	eErrorID		:= fbReadInputRegistersFc04.eErrorID;
	eExeptionCode	:= fbReadInputRegistersFc04.eException;
END_IF;
(* Write Single Coil Fc05 Error *)
IF fbWriteSingleCoilFc05.xError AND NOT xErrorHappen THEN
	xErrorHappen 	:= fbWriteSingleCoilFc05.xError;
	eErrorID		:= fbWriteSingleCoilFc05.eErrorID;
	eExeptionCode	:= fbWriteSingleCoilFc05.eException;
END_IF;
(* Write Single Register Fc06 Error *)
IF fbWriteSingleRegisterFc06.xError AND NOT xErrorHappen THEN
	xErrorHappen 	:= fbWriteSingleRegisterFc06.xError;
	eErrorID		:= fbWriteSingleRegisterFc06.eErrorID;
	eExeptionCode	:= fbWriteSingleRegisterFc06.eException;
END_IF;		
(* Write Multiple Coils Fc15 Error *)
IF fbWriteMultipleCoilsFc15.xError AND NOT xErrorHappen THEN
	xErrorHappen 	:= fbWriteMultipleCoilsFc15.xError;
	eErrorID		:= fbWriteMultipleCoilsFc15.eErrorID;
	eExeptionCode	:= fbWriteMultipleCoilsFc15.eException;
END_IF;
(* Write Multiple Registers Fc16 Error *)
IF fbWriteMultipleRegistersFc16.xError AND NOT xErrorHappen THEN
	xErrorHappen 	:= fbWriteMultipleRegistersFc16.xError;
	eErrorID		:= fbWriteMultipleRegistersFc16.eErrorID;
	eExeptionCode	:= fbWriteMultipleRegistersFc16.eException;
END_IF;
END_ACTION

END_FUNCTION_BLOCK

// 30 Program Organization Units/CLIENT/TCP/FB_MB_CLIENT_TCP_1
FUNCTION_BLOCK FB_MB_CLIENT_TCP_1 EXTENDS FB_MB_CLIENT IMPLEMENTS ITF_MB_CLIENT_TCP
VAR_OUTPUT
END_VAR
VAR
	(* Config *)
	fbConfigFile				:	CtaSysConfig.fbConfigFile;
	scParameter                	: 	scTcpClientParameter;
END_VAR

(* Config File *)
actConfig();

ACTION actConfig:
(* Config File *)
fbConfigFile();

scParameter.fbxEnable		(_usiParaNr := 1,itfConfigFb := fbConfigFile										);		
scParameter.fbusiNodeId		(_usiParaNr := 2,itfConfigFb := fbConfigFile,_MinInit := 0	  , _MaxInit := 255		);		
scParameter.fbtTimeOut		(_usiParaNr := 3,itfConfigFb := fbConfigFile,_MinInit := T#0MS, _MaxInit := T#5M 	);		
scParameter.fbtReadDelay	(_usiParaNr := 4,itfConfigFb := fbConfigFile,_MinInit := T#0MS, _MaxInit := T#5M 	);		
scParameter.fbtWriteDelay	(_usiParaNr := 5,itfConfigFb := fbConfigFile,_MinInit := T#0MS, _MaxInit := T#5M 	);	
scParameter.fbuiPort		(_usiParaNr := 6,itfConfigFb := fbConfigFile										);
scParameter.fbstIpAdress	(_usiParaNr := 7,itfConfigFb := fbConfigFile										);

(* Check Ip *)
IF scParameter.fbstIpAdress.proStateChanged THEN
	IF NOT fcCheckIp(scParameter.fbstIPAdress.proValue) THEN
		fcSetInitialIPString(scParameter.fbstIpAdress);
	END_IF;
END_IF;
END_ACTION

PROPERTY ENABLE : BOOL
GET
ENABLE := scParameter.fbxEnable.proValue;
END_GET
END_PROPERTY

PROPERTY IP_ADRESS : STRING(15)
GET
IP_ADRESS := scParameter.fbstIpAdress.proValue;
END_GET
END_PROPERTY

PROPERTY P_fbtReadDelay : CtaSysConfig.ITF_DATATYPE
GET
P_fbtReadDelay := scParameter.fbtReadDelay;
END_GET
END_PROPERTY

PROPERTY P_fbtTimeOut : CtaSysConfig.ITF_DATATYPE
GET
P_fbtTimeOut := scParameter.fbtTimeOut;
END_GET
END_PROPERTY

PROPERTY P_fbtWriteDelay : CtaSysConfig.ITF_DATATYPE
GET
P_fbtWriteDelay := scParameter.fbtWriteDelay;
END_GET
END_PROPERTY

PROPERTY P_fbuiPort : CtaSysConfig.ITF_DATATYPE
GET
P_fbuiPort := scParameter.fbuiPort;
END_GET
END_PROPERTY

PROPERTY P_fbusiNodeId : CtaSysConfig.ITF_DATATYPE
GET
P_fbusiNodeId := scParameter.fbusiNodeId;
END_GET
END_PROPERTY

PROPERTY P_fbxEnable : CtaSysConfig.ITF_DATATYPE
GET
P_fbxEnable := scParameter.fbxEnable;
END_GET
END_PROPERTY

PROPERTY WRITE_DELAY : TIME
GET
WRITE_DELAY := scParameter.fbtWriteDelay.proValue;
END_GET
END_PROPERTY

PROPERTY PORT : UINT
GET
PORT := scParameter.fbuiPort.proValue;
END_GET
END_PROPERTY

PROPERTY NODE_ID : USINT
GET
NODE_ID := scParameter.fbusiNodeId.proValue;
END_GET
END_PROPERTY

PROPERTY P_fbstIpAdress : CtaSysConfig.ITF_DATATYPE
GET
P_fbstIpAdress := scParameter.fbstIpAdress;
END_GET
END_PROPERTY

PROPERTY READ_DELAY : TIME
GET
READ_DELAY := scParameter.fbtReadDelay.proValue;
END_GET
END_PROPERTY

PROPERTY TIMEOUT : TIME
GET
TIMEOUT := scParameter.fbtTimeOut.proValue;
END_GET
END_PROPERTY

END_FUNCTION_BLOCK

// 40 Visualizations/SERVER/SERIAL/VIS_SERVER_SERIAL_STATE
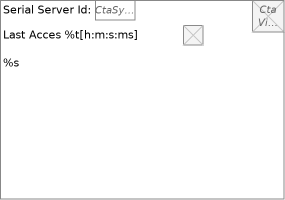
VISUALIZATION VIS_SERVER_SERIAL_STATE  // 285x200
VAR_INPUT
	ITF_SERVER_INFO_PARA_IN : ITF_SERVER_INFO_PARA;
END_VAR
    Frame (0,0 285x200), invisible if: NOT __QUERYINTERFACE(ITF_SERVER_INFO_PARA_IN,ITF_SERVER_INFO_PARA_IN)
        shows VIS_SERVER_SERIAL_STATE_INFO(ITF_SERVER_INFO_PARA_IN := ITF_SERVER_INFO_PARA_IN)
END_VISUALIZATION

// 40 Visualizations/CLIENT/CLIENT/DIA_CLIENT
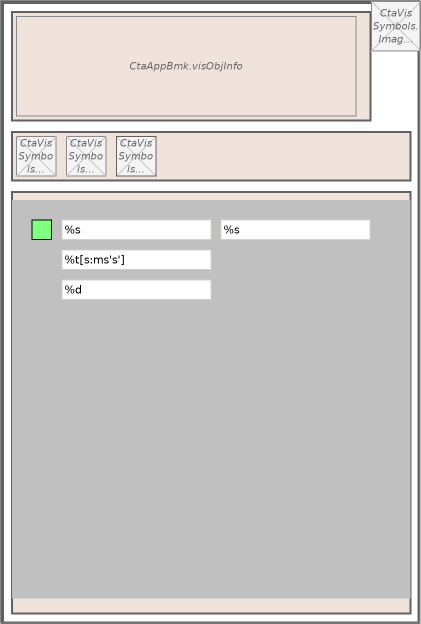
VISUALIZATION DIA_CLIENT  // 421x624
VAR_INPUT
	ITF_CLIENT_IN : ITF_CLIENT;
END_VAR
VAR
	uiPopUpGruppe 			:	UINT;
END_VAR
    RoundedRectangle (1,1 419x623)
    RoundedRectangle (11,11 360x110)
    RoundedRectangle (11,191 400x423)
    RoundedRectangle (11,131 400x50)
    Frame (16,16 340x100)
        shows CtaAppBmk.visObjInfo(ITF_BMK_IN := ITF_CLIENT_IN)
    Image (371,1 50x50), image: CtaVisSymbols.ImagePool.close_solo_black
        OnMouseClick:  Dialog=Current Dialog, Result=OK, NumpadKeypadSet=True
    Frame (11,136 400x40)
        shows VIS_CLIENT_MENÜ(uiPopUpGruppe := uiPopUpGruppe)
    Frame (12,200 398x400), frame switch variable: uiPopUpGruppe
        shows VIS_CLIENT_OVERWIEV(ITF_CLIENT_IN := ITF_CLIENT_IN)
        shows VIS_CLIENT_PARAMETER(ITF_CLIENT_IN := ITF_CLIENT_IN)
        shows VIS_CLIENT_JOBS(ITF_CLIENT_IN := ITF_CLIENT_IN)
    InvisibleInput (0,0 371x50)
END_VISUALIZATION

// 40 Visualizations/SERVER/SERIAL/VIS_SERVER_SERIAL_STATE_INFO
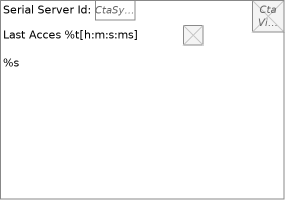
VISUALIZATION VIS_SERVER_SERIAL_STATE_INFO  // 285x200
VAR_INPUT
	ITF_SERVER_INFO_PARA_IN : ITF_SERVER_INFO_PARA;
END_VAR
    Label (0,0 96x20), "Serial Server Id:"
    Frame (95,0 40x20)
        shows CtaSysConfig.visUSINT(visfbUSINTIn := ITF_SERVER_INFO_PARA_IN.P_Serial_fbusiNodeId)
    Textfield (0,55 285x144), "%s", text variable: ITF_SERVER_INFO_PARA_IN.RequestDataSerial
    Textfield (0,25 178x20), "Last Acces %t[h:m:s:ms]", text variable: ITF_SERVER_INFO_PARA_IN.NoSerialAccesSince
    Image (183,25 20x20), invisible if: NOT ITF_SERVER_INFO_PARA_IN.TimeOutSerialWatchDog, image: CtaVisSymbols.ImagePool.CtaError
    Image (252,0 32x32), image: CtaVisSymbols.ImagePool.gear
        OnMouseClick:  Dialog=DIA_SERVER_SERIAL_PARAMETER, Parameters={ITF_SERVER_INFO_PARA_IN: ITF_SERVER_INFO_PARA_IN}, OpenCentered=True
END_VISUALIZATION

// 40 Visualizations/CLIENT/CLIENT/JOBS/VIS_CLIENT_JOBS
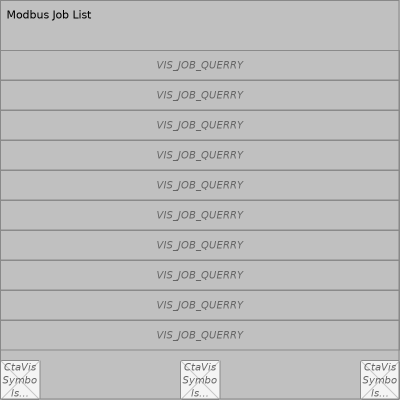
VISUALIZATION VIS_CLIENT_JOBS  // 400x400
VAR_INPUT
	ITF_CLIENT_IN : ITF_CLIENT;	
END_VAR
    Frame (0,0 400x400), invisible if: NOT __QUERYINTERFACE(ITF_CLIENT_IN,ITF_CLIENT_IN)
        shows VIS_CLIENT_JOBS_QUERRY(ITF_CLIENT_IN := ITF_CLIENT_IN)
END_VISUALIZATION

// 40 Visualizations/CLIENT/CLIENT/JOBS/VIS_CLIENT_JOBS_QUERRY
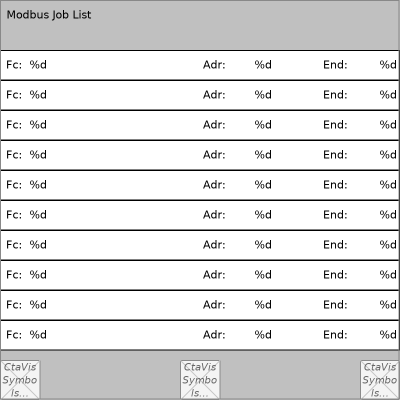
VISUALIZATION VIS_CLIENT_JOBS_QUERRY  // 400x400
VAR_INPUT
	ITF_CLIENT_IN : ITF_CLIENT;
END_VAR
    Rectangle (0,0 400x400)
    Frame (0,50 400x300)
        shows VIS_CLIENT_JOBS_TABLE(AY_ITF_MBJOB := ITF_CLIENT_IN.AY_ITF_MBJOB_VIS)
    Image (360,360 40x40), image: CtaVisSymbols.ImagePool.arrow-right_square
        OnMouseClick: execute { ITF_CLIENT_IN.RELOAD_ARRAY(FALSe,TRUE,FALSE); }
    Image (0,360 40x40), image: CtaVisSymbols.ImagePool.arrow-left_square
        OnMouseClick: execute { ITF_CLIENT_IN.RELOAD_ARRAY(FALSe,FALse,TRUE); }
    Image (180,360 40x40), image: CtaVisSymbols.ImagePool.refresh
        OnMouseClick: execute { ITF_CLIENT_IN.RELOAD_ARRAY(TRUE,FALSE,FALSE); }
    Label (0,0 200x30), "Modbus Job List"
END_VISUALIZATION

// 40 Visualizations/CLIENT/CLIENT/JOBS/VIS_CLIENT_JOBS_TABLE
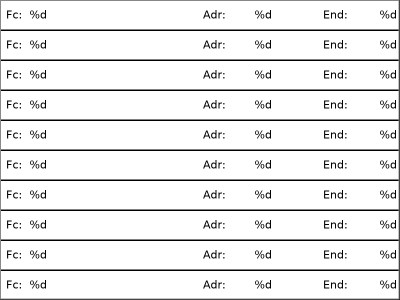
VISUALIZATION VIS_CLIENT_JOBS_TABLE  // 400x300
VAR_INPUT
	AY_ITF_MBJOB	:	ARRAY[0..9] OF ITF_MBJOB;
END_VAR
    Frame (0,0 400x30)
        shows VIS_JOB(ITF_MBJOBIN := AY_ITF_MBJOB[0])
    Frame (0,30 400x30)
        shows VIS_JOB(ITF_MBJOBIN := AY_ITF_MBJOB[1])
    Frame (0,60 400x30)
        shows VIS_JOB(ITF_MBJOBIN := AY_ITF_MBJOB[2])
    Frame (0,90 400x30)
        shows VIS_JOB(ITF_MBJOBIN := AY_ITF_MBJOB[3])
    Frame (0,120 400x30)
        shows VIS_JOB(ITF_MBJOBIN := AY_ITF_MBJOB[4])
    Frame (0,150 400x30)
        shows VIS_JOB(ITF_MBJOBIN := AY_ITF_MBJOB[5])
    Frame (0,180 400x30)
        shows VIS_JOB(ITF_MBJOBIN := AY_ITF_MBJOB[6])
    Frame (0,210 400x30)
        shows VIS_JOB(ITF_MBJOBIN := AY_ITF_MBJOB[7])
    Frame (0,240 400x30)
        shows VIS_JOB(ITF_MBJOBIN := AY_ITF_MBJOB[8])
    Frame (0,270 400x30)
        shows VIS_JOB(ITF_MBJOBIN := AY_ITF_MBJOB[9])
END_VISUALIZATION

// 40 Visualizations/CLIENT/CLIENT/MENÜ/VIS_CLIENT_MENÜ
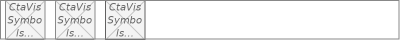
VISUALIZATION VIS_CLIENT_MENÜ  // 400x40
VAR_IN_OUT
	uiPopUpGruppe 			:	UINT;
END_VAR
    Rectangle (100,0 40x40), colour toggle: uiPopUpGruppe = 2
        OnMouseDown: execute { uiPopUpGruppe := 2; }
    Group (5,0 40x40)
        RoundedRectangle (0,0 40x40), colour toggle: uiPopUpGruppe = 0
            OnMouseDown: execute { uiPopUpGruppe := 0; }
        Image (0,0 40x40), image: CtaVisSymbols.ImagePool.eye
            OnMouseDown: execute { uiPopUpGruppe := 0; }
    Group (55,0 40x40)
        RoundedRectangle (0,0 40x40), colour toggle: uiPopUpGruppe = 2
            OnMouseDown: execute { uiPopUpGruppe := 1; }
        Image (0,0 40x40), image: CtaVisSymbols.ImagePool.gear
            OnMouseDown: execute { uiPopUpGruppe := 1; }
    Group (105,0 40x40)
        Image (0,0 40x40), image: CtaVisSymbols.ImagePool.lan
            OnMouseDown: execute { uiPopUpGruppe := 2; }
        RoundedRectangle (0,0 40x40), colour toggle: uiPopUpGruppe = 2
            OnMouseDown: execute { uiPopUpGruppe := 2; }
END_VISUALIZATION

// 40 Visualizations/CLIENT/CLIENT/OVERWIEV/VIS_CLIENT_OVERWIEV
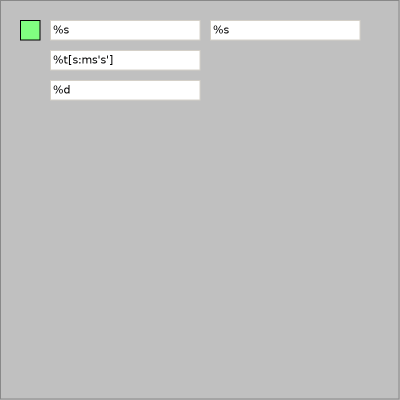
VISUALIZATION VIS_CLIENT_OVERWIEV  // 400x400
VAR_INPUT
	ITF_CLIENT_IN : ITF_CLIENT;	
END_VAR
    Frame (0,0 400x400), invisible if: NOT __QUERYINTERFACE(ITF_CLIENT_IN,ITF_CLIENT_IN)
        shows VIS_CLIENT_OVERWIEV_QUERY(ITF_CLIENT_IN := ITF_CLIENT_IN)
END_VISUALIZATION

// 40 Visualizations/CLIENT/CLIENT/OVERWIEV/VIS_CLIENT_OVERWIEV_QUERY
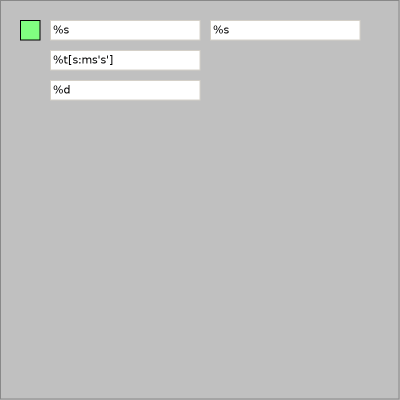
VISUALIZATION VIS_CLIENT_OVERWIEV_QUERY  // 400x400
VAR_INPUT
	ITF_CLIENT_IN : ITF_CLIENT;	
END_VAR
    Rectangle (0,0 400x400)
    Rectangle (20,20 20x20), colour toggle: ITF_CLIENT_IN.ERROR
    Textfield (50,20 150x20), "%s", text variable: TO_STRING(ITF_CLIENT_IN.ERROR_ID)
    Textfield (210,20 150x20), "%s", text variable: TO_STRING(ITF_CLIENT_IN.EXEPTION_CODE)
    Textfield (50,50 150x20), "%t[s:ms's']", text variable: ITF_CLIENT_IN.ExecuteTime
    Textfield (50,80 150x20), "%d", text variable: ITF_CLIENT_IN.COUNT
END_VISUALIZATION

// 40 Visualizations/CLIENT/CLIENT/PARAMETER/VIS_CLIENT_PARAMETER
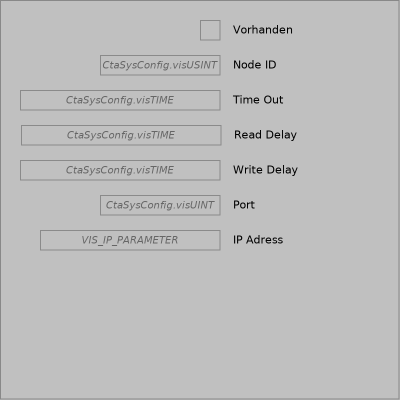
VISUALIZATION VIS_CLIENT_PARAMETER  // 400x400
VAR_INPUT
	ITF_CLIENT_IN : ITF_CLIENT;	
END_VAR
    Rectangle (0,0 400x400)
    Frame (0,0 400x400)
        shows VIS_CLIENT_PARAMETER_RTU(ITF_CLIENT_IN := ITF_CLIENT_IN)
    Frame (0,0 400x400), invisible if: NOT __QUERYINTERFACE(ITF_CLIENT_IN,ITF_CLIENT_IN)
        shows VIS_CLIENT_PARAMETER_TCP(ITF_CLIENT_IN := ITF_CLIENT_IN)
END_VISUALIZATION

// 40 Visualizations/CLIENT/RTU/PARAMETER/VIS_CLIENT_PARAMETER_RTU_QUERY
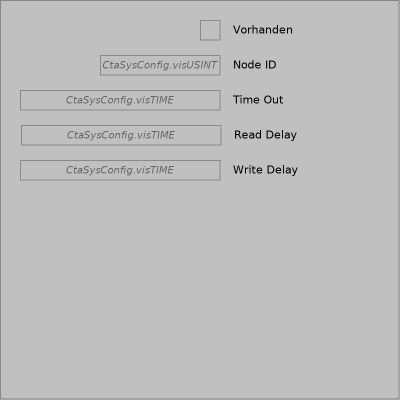
VISUALIZATION VIS_CLIENT_PARAMETER_RTU_QUERY  // 400x400
VAR_INPUT
	ITF_MB_CLIENT_RTU_IN : ITF_MB_CLIENT_RTU;	
END_VAR
    Rectangle (0,0 400x400)
    Frame (200,20 20x20)
        shows CtaSysConfig.visBOOL(visfbBOOLIn := ITF_MB_CLIENT_RTU_IN.P_fbxEnable)
    Label (230,20 150x20), "Vorhanden"
    Label (230,55 150x20), "Node ID"
    Frame (100,55 120x20)
        shows CtaSysConfig.visUSINT(visfbUSINTIn := ITF_MB_CLIENT_RTU_IN.P_fbusiNodeId)
    Label (230,90 150x20), "Time Out"
    Frame (20,90 200x20)
        shows CtaSysConfig.visTIME(visfbTIMEIn := ITF_MB_CLIENT_RTU_IN.P_fbtTimeOut)
    Frame (21,125 200x20)
        shows CtaSysConfig.visTIME(visfbTIMEIn := ITF_MB_CLIENT_RTU_IN.P_fbtReadDelay)
    Label (231,125 150x20), "Read Delay"
    Frame (20,160 200x20)
        shows CtaSysConfig.visTIME(visfbTIMEIn := ITF_MB_CLIENT_RTU_IN.P_fbtWriteDelay)
    Label (230,160 150x20), "Write Delay"
END_VISUALIZATION

// 40 Visualizations/CLIENT/RTU/PARAMETER/VIS_CLIENT_PARAMETER_RTU
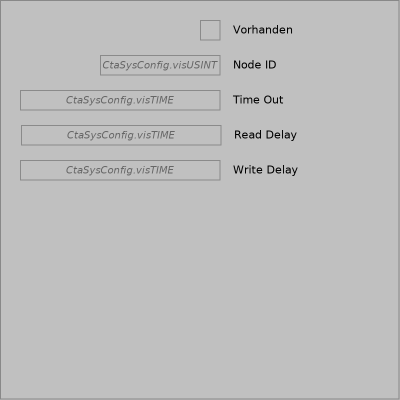
VISUALIZATION VIS_CLIENT_PARAMETER_RTU  // 400x400
VAR_INPUT
	ITF_CLIENT_IN : ITF_CLIENT;	
END_VAR
VAR
	ITF_MB_CLIENT_RTU_QUERY	:	ITF_MB_CLIENT_RTU;
END_VAR
    Frame (0,0 400x400), invisible if: NOT __QUERYINTERFACE(ITF_CLIENT_IN,ITF_MB_CLIENT_RTU_QUERY)
        shows VIS_CLIENT_PARAMETER_RTU_TEMP(ITF_MB_CLIENT_RTU_QUERY := ITF_MB_CLIENT_RTU_QUERY)
END_VISUALIZATION

// 40 Visualizations/CLIENT/RTU/PARAMETER/VIS_CLIENT_PARAMETER_RTU_TEMP
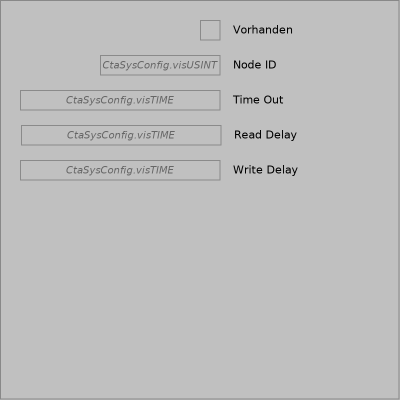
VISUALIZATION VIS_CLIENT_PARAMETER_RTU_TEMP  // 400x400
VAR_INPUT
	ITF_MB_CLIENT_RTU_QUERY	:	ITF_MB_CLIENT_RTU;
END_VAR
    Frame (0,0 400x400), invisible if: NOT __QUERYINTERFACE(ITF_MB_CLIENT_RTU_QUERY,ITF_MB_CLIENT_RTU_QUERY)
        shows VIS_CLIENT_PARAMETER_RTU_QUERY(ITF_MB_CLIENT_RTU_IN := ITF_MB_CLIENT_RTU_QUERY)
END_VISUALIZATION

// 40 Visualizations/CLIENT/TCP/PARAMETER/VIS_CLIENT_PARAMETER_TCP
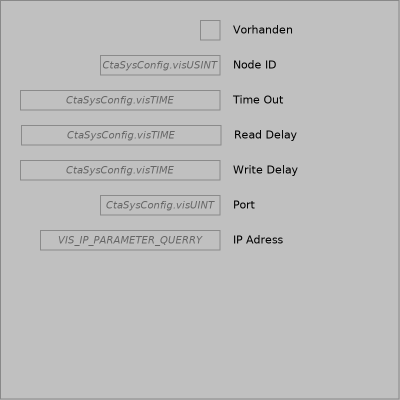
VISUALIZATION VIS_CLIENT_PARAMETER_TCP  // 400x400
VAR_INPUT
	ITF_CLIENT_IN : ITF_CLIENT;	
END_VAR
VAR
	ITF_MB_CLIENT_TCP_QUERY	:	ITF_MB_CLIENT_TCP;
END_VAR
    Frame (0,0 400x400), invisible if: NOT __QUERYINTERFACE(ITF_CLIENT_IN,ITF_MB_CLIENT_TCP_QUERY)
        shows VIS_CLIENT_PARAMETER_TCP_TEMP(ITF_MB_CLIENT_TCP_QUERY := ITF_MB_CLIENT_TCP_QUERY)
END_VISUALIZATION

// 40 Visualizations/CLIENT/TCP/PARAMETER/VIS_CLIENT_PARAMETER_TCP_TEMP
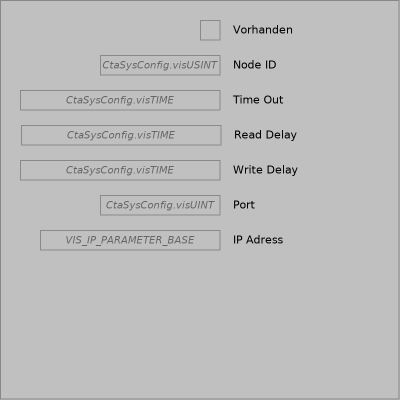
VISUALIZATION VIS_CLIENT_PARAMETER_TCP_TEMP  // 400x400
VAR_INPUT
	ITF_MB_CLIENT_TCP_QUERY	:	ITF_MB_CLIENT_TCP;
END_VAR
    Frame (0,0 400x400), invisible if: NOT __QUERYINTERFACE(ITF_MB_CLIENT_TCP_QUERY,ITF_MB_CLIENT_TCP_QUERY)
        shows VIS_CLIENT_PARAMETER_TCP_QUERY(ITF_MB_CLIENT_TCP_IN := ITF_MB_CLIENT_TCP_QUERY)
END_VISUALIZATION

// 40 Visualizations/CLIENT/TCP/PARAMETER/VIS_CLIENT_PARAMETER_TCP_QUERY
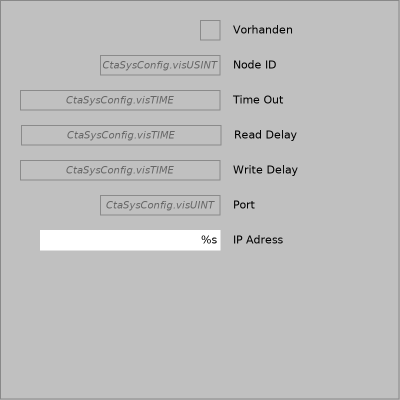
VISUALIZATION VIS_CLIENT_PARAMETER_TCP_QUERY  // 400x400
VAR_INPUT
	ITF_MB_CLIENT_TCP_IN : ITF_MB_CLIENT_TCP;	
END_VAR
    Rectangle (0,0 400x400)
    Frame (200,20 20x20)
        shows CtaSysConfig.visBOOL(visfbBOOLIn := ITF_MB_CLIENT_TCP_IN.P_fbxEnable)
    Label (230,20 150x20), "Vorhanden"
    Label (230,55 150x20), "Node ID"
    Frame (100,55 120x20)
        shows CtaSysConfig.visUSINT(visfbUSINTIn := ITF_MB_CLIENT_TCP_IN.P_fbusiNodeId)
    Label (230,90 150x20), "Time Out"
    Frame (20,90 200x20)
        shows CtaSysConfig.visTIME(visfbTIMEIn := ITF_MB_CLIENT_TCP_IN.P_fbtTimeOut)
    Frame (21,125 200x20)
        shows CtaSysConfig.visTIME(visfbTIMEIn := ITF_MB_CLIENT_TCP_IN.P_fbtReadDelay)
    Label (231,125 150x20), "Read Delay"
    Frame (20,160 200x20)
        shows CtaSysConfig.visTIME(visfbTIMEIn := ITF_MB_CLIENT_TCP_IN.P_fbtWriteDelay)
    Label (230,160 150x20), "Write Delay"
    Label (230,195 150x20), "Port"
    Frame (100,195 120x20)
        shows CtaSysConfig.visUINT(visfbUINTIn := ITF_MB_CLIENT_TCP_IN.P_fbuiPort)
    Label (230,230 150x20), "IP Adress"
    Frame (40,230 180x20)
        shows VIS_IP_PARAMETER(ITF_DATATYPE_IN := ITF_MB_CLIENT_TCP_IN.P_fbstIpAdress)
END_VISUALIZATION

// 40 Visualizations/CLIENTMANAGER/DIA_CLIENT_MANAGER
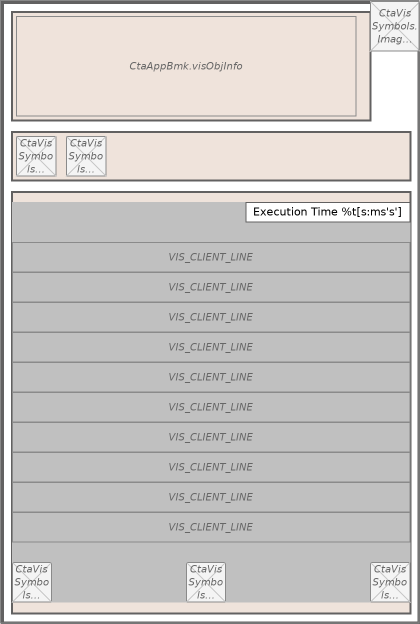
VISUALIZATION DIA_CLIENT_MANAGER  // 420x624
VAR_INPUT
	ITF_CLIENT_MANAGER_IN : ITF_MB_CLIENTMANAGER;
END_VAR
VAR
	uiPopUpGruppe 			:	UINT;
END_VAR
    RoundedRectangle (1,1 419x623)
    RoundedRectangle (11,11 360x110)
    RoundedRectangle (11,191 400x423)
    RoundedRectangle (11,131 400x50)
    Image (370,1 50x50), image: CtaVisSymbols.ImagePool.close_solo_black
        OnMouseClick:  Dialog=Current Dialog, Result=OK, NumpadKeypadSet=True
    Frame (16,16 340x100)
        shows CtaAppBmk.visObjInfo(ITF_BMK_IN := ITF_CLIENT_MANAGER_IN)
    Frame (11,136 400x40)
        shows VIS_CLIENTMANAGER_MENÜ(uiPopUpGruppe := uiPopUpGruppe)
    Frame (12,202 398x400), invisible if: NOT __QUERYINTERFACE(ITF_CLIENT_MANAGER_IN,ITF_CLIENT_MANAGER_IN), frame switch variable: uiPopUpGruppe
        shows VIS_CLIENT_MANAGER_OVERWIEV(ITF_CLIENT_MANAGER_IN := ITF_CLIENT_MANAGER_IN)
        shows VIS_CLIENT_MANAGER_PARAMETER(ITF_CLIENT_MANAGER_IN := ITF_CLIENT_MANAGER_IN)
    InvisibleInput (0,0 371x50)
END_VISUALIZATION

// 40 Visualizations/CLIENTMANAGER/LINE/VIS_CLIENT_LINE
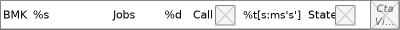
VISUALIZATION VIS_CLIENT_LINE  // 400x30
VAR_INPUT
	ITF_CLIENTIN		:	ITF_CLIENT;
END_VAR
    Frame (0,0 400x30), invisible if: NOT __QUERYINTERFACE(ITF_CLIENTIN,ITF_CLIENTIN)
        shows VIS_CLIENT_LINE_QUERRY(ITF_CLIENTIN := ITF_CLIENTIN)
END_VISUALIZATION

// 40 Visualizations/CLIENTMANAGER/LINE/VIS_CLIENT_LINE_QUERRY
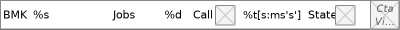
VISUALIZATION VIS_CLIENT_LINE_QUERRY  // 400x30
VAR_INPUT
	ITF_CLIENTIN		:	ITF_CLIENT;
END_VAR
    Rectangle (0,0 400x30)
    RoundedRectangle (0,0 400x30)
    Textfield (240,0 60x30), "%t[s:ms's']", text variable: ITF_CLIENTIN.ExecuteTime
    Textfield (0,0 30x30), "BMK"
    Textfield (30,0 75x30), "%s", text variable: ITF_CLIENTIN.proGetBMK
    Textfield (145,0 40x30), "%d", text variable: ITF_CLIENTIN.COUNT
    Textfield (110,0 30x30), "Jobs"
    Textfield (190,0 35x30), "Call"
    Textfield (305,0 35x30), "State"
    Image (335,5 20x20), invisible if: NOT ITF_CLIENTIN.ERROR, image: CtaVisSymbols.ImagePool.CtaError
    Image (215,5 20x20), invisible if: NOT ITF_CLIENTIN.IsCurrentCall, image: CtaVisSymbols.ImagePool.check_green
    Image (370,0 30x30), image: CtaVisSymbols.ImagePool.gear
        OnMouseClick:  Dialog=DIA_CLIENT, Parameters={ITF_CLIENT_IN: ITF_CLIENTIN}, OpenModal=True, OpenCentered=True
    Image (335,5 20x20), invisible if: ITF_CLIENTIN.ERROR, image: CtaVisSymbols.ImagePool.check_green
END_VISUALIZATION

// 40 Visualizations/CLIENTMANAGER/MENÜ/VIS_CLIENTMANAGER_MENÜ
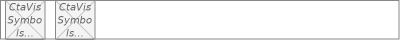
VISUALIZATION VIS_CLIENTMANAGER_MENÜ  // 400x40
VAR_IN_OUT
	uiPopUpGruppe 			:	UINT;
END_VAR
    Group (5,0 40x40)
        RoundedRectangle (0,0 40x40), colour toggle: uiPopUpGruppe = 0
            OnMouseDown: execute { uiPopUpGruppe := 0; }
        Image (0,0 40x40), image: CtaVisSymbols.ImagePool.eye
            OnMouseDown: execute { uiPopUpGruppe := 0; }
    Group (55,0 40x40)
        RoundedRectangle (0,0 40x40), colour toggle: uiPopUpGruppe = 1
            OnMouseDown: execute { uiPopUpGruppe := 1; }
        Image (0,0 40x40), image: CtaVisSymbols.ImagePool.gear
            OnMouseDown: execute { uiPopUpGruppe := 1; }
END_VISUALIZATION

// 40 Visualizations/CLIENTMANAGER/TCP/PARAMETER/VIS_CLIENT_MANAGER_PARAMETER_TCP
VISUALIZATION VIS_CLIENT_MANAGER_PARAMETER_TCP  // 400x400
VAR_INPUT
	ITF_CLIENT_MANAGER_IN : ITF_MB_CLIENTMANAGER;	
END_VAR
VAR
	ITF_CLIENT_MANAGER_TCP_IN : ITF_MB_CLIENTMANAGER_TCP;	
END_VAR
    Frame (0,0 400x400), invisible if: NOT __QUERYINTERFACE(ITF_CLIENT_MANAGER_IN,ITF_CLIENT_MANAGER_TCP_IN)
        shows VIS_CLIENT_MANAGER_PARAMETER_TCP_QUERY(ITF_CLIENT_MANAGER_TCP_IN := ITF_CLIENT_MANAGER_TCP_IN)
END_VISUALIZATION

// 40 Visualizations/CLIENTMANAGER/TCP/PARAMETER/VIS_CLIENT_MANAGER_PARAMETER_TCP_QUERY
VISUALIZATION VIS_CLIENT_MANAGER_PARAMETER_TCP_QUERY  // 400x400
VAR_INPUT
	ITF_CLIENT_MANAGER_TCP_IN : ITF_MB_CLIENTMANAGER_TCP;	
END_VAR
END_VISUALIZATION

// 40 Visualizations/HELPER/VIS_IP_PARAMETER
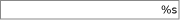
VISUALIZATION VIS_IP_PARAMETER  // 180x20
VAR_INPUT
    ITF_DATATYPE_IN : CtaSysConfig.ITF_DATATYPE;	
END_VAR
VAR
	ITF_STRING40In : CtaSysConfig.ITF_STRING40;	
END_VAR
    Frame (0,0 180x20), invisible if: NOT __QUERYINTERFACE(ITF_DATATYPE_IN,ITF_STRING40In), input disabled if: NOT __QUERYINTERFACE(ITF_DATATYPE_IN,ITF_STRING40In)
        shows VIS_IP_PARAMETER_QUERRY(ITF_STRING40In := ITF_STRING40In)
END_VISUALIZATION

// 40 Visualizations/HELPER/DIA_IP_INPUT
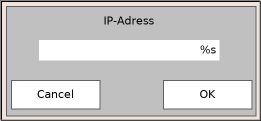
VISUALIZATION DIA_IP_INPUT  // 261x121
VAR_INPUT
    ITF_STRING40In : CtaSysConfig.ITF_STRING40;	
END_VAR
VAR
	stIPTemp    :   STRING;
END_VAR
    RoundedRectangle (1,1 260x120)
    RoundedRectangle (6,6 250x110)
    Textfield (39,40 180x20), "%s", text variable: stIPTemp
        OnMouseClick: write the text variable via Default
    RoundedRectangle (11,80 89x29), "Cancel"
        OnMouseClick:  Dialog=Current Dialog, Result=Cancel, NumpadKeypadSet=True
    RoundedRectangle (163,80 89x29), "OK"
        OnMouseClick: execute {
            IF fcCheckIp(stIPTemp) THEN
                ITF_STRING40In.proValue := stIPTemp;
            ELSE
                ITF_STRING40In.proValue := 'Wrong IP';
            END_IF
        }
        OnMouseClick:  Dialog=Current Dialog, Result=OK, NumpadKeypadSet=True
    Label (39,6 180x30), "IP-Adress"
END_VISUALIZATION

// 40 Visualizations/HELPER/VIS_IP_PARAMETER_QUERRY
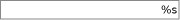
VISUALIZATION VIS_IP_PARAMETER_QUERRY  // 180x20
VAR_INPUT
    ITF_STRING40In : CtaSysConfig.ITF_STRING40;	
END_VAR
    Frame (0,0 180x20), invisible if: NOT __QUERYINTERFACE(ITF_STRING40In,ITF_STRING40In), input disabled if: NOT __QUERYINTERFACE(ITF_STRING40In,ITF_STRING40In)
        shows VIS_IP_PARAMETER_BASE(ITF_STRING40In := ITF_STRING40In)
END_VISUALIZATION

// 40 Visualizations/HELPER/VIS_IP_PARAMETER_BASE
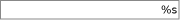
VISUALIZATION VIS_IP_PARAMETER_BASE  // 180x20
VAR_INPUT
    ITF_STRING40In : CtaSysConfig.ITF_STRING40;	
END_VAR
    Textfield (0,0 180x20), "%s", text variable: ITF_STRING40In.proValue, invisible if: NOT fcSetInitialIPString(ITF_STRING40In)
        OnMouseClick:  Dialog=DIA_IP_INPUT, Parameters={stIPTemp: , ITF_STRING40In: ITF_STRING40In}, OpenModal=True, OpenCentered=True
END_VISUALIZATION

// 40 Visualizations/MBJOB/VIS_JOB
